KUKA KRL program: EPS_2_25694_WD06A_A_20260120031700.src

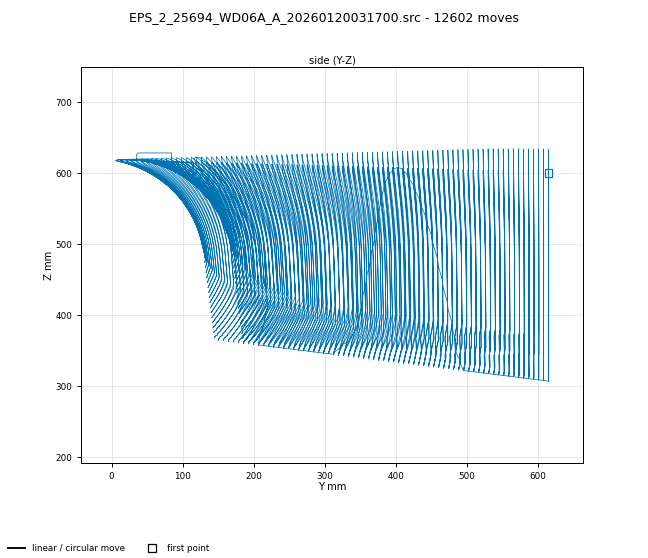
[picture p0: tool path of EPS_2_25694_WD06A_A_20260120031700.src, 12602 of 12604 moves have a stored position in this frame; points joined in program order, loops and branches not executed]
&ACCESS RVP
&REL 4
&COMMENT QRS 19112012
&PARAM EDITMASK = *
DEF PART()
EXT BAS (BAS_COMMAND :IN,REAL :IN )
INT I
BAS (#INITMOV,0 )

;KUKA QRS Post kuka4.cps  Date:22-06-2017 !

File_ID=2995

QRS_PRE_INIT()

;Init var - Until changes are made in qrs_pre_init
Outlet_Square_prg=0
Inlet_1_Square_prg=0
Inlet_2_Square_prg=0
Inlet_3_Square_prg=0
Inlet_4_Square_prg=0
Inlet_5_Square_prg=0

Outlet_1={X 0.000, Y 527.380, Z 509.000, B 0.000, E1 0.000 }
Inlet_1={X 0.000, Y 529.540, Z 479.000, B 0.000, E1 174.000 }
Outlet_1_type=251
Inlet_1_type=251
;QRS#1=Sidecore dimensions
;QRS#2=250-10" PVC SDR 35
;QRS#3=250-10" PVC SDR 35
;QRS#4=
;QRS#5=
;QRS#6=
;QRS#7=
;QRS#8=
;QRS#9=14M PSX
;QRS#10=14M PSX
;QRS#11=
;QRS#12=
;QRS#13=
;QRS#14=
;QRS#15=
;QRS#16=1220x127x914 3'
;QRS#17=EPS Height
;QRS#18=634,5
;QRS#19=*
;QRS#20= UPDATED VERSION 22-06-2017
;QRS#21=*
Outlet_Square=0100
Inlet_1_Square=0100
Inlet_2_Square=0
Inlet_3_Square=0
Inlet_4_Square=0
Inlet_5_Square=0
Mill_Square=1
Outlet_Square_Prg=205
Inlet_1_Square_prg=205

QRS_INIT()

$ADVANCE=5

; T1
PTP {E1 173.639,E2 173.639}
PTP {X 0,Y 615.429,A -85,B 0,C 180,E1 173.639,E2 173.639,E3 0,E4 0,E5 0,E6 0}
QRS_SPEED_INIT()
LIN {X 0,Y 615.429,Z 600,A -85,B 0,C 180,E1 173.639,E2 173.639,E3 0,E4 0,E5 0,E6 0} C_VEL
LIN {X 0,Y 615.429,Z 317.5,A -85,B 0,C 180,E1 173.639,E2 173.639} C_VEL
LIN {X 0,Y 615.429,Z 309.322,A -85,B 0,C 180,E1 173.639,E2 173.639} C_VEL
LIN {X 0,Y 615.432,Z 307.322,A -85,B 0,C 180,E1 173.453,E2 173.453} C_VEL
LIN {X 0,Y 615.494,Z 307.326,A -85,B 0,C 180,E1 170.801,E2 170.801} C_VEL
LIN {X 0,Y 615.451,Z 307.317,A -85,B 0,C 180,E1 168.138,E2 168.138} C_VEL
LIN {X 0,Y 615.446,Z 307.318,A -85,B 0,C 180,E1 166.077,E2 166.077} C_VEL
LIN {X 0,Y 615.443,Z 307.321,A -85,B 0,C 180,E1 163.578,E2 163.578} C_VEL
LIN {X 0,Y 615.461,Z 307.322,A -85,B 0,C 180,E1 161.353,E2 161.353} C_VEL
LIN {X 0,Y 615.492,Z 307.312,A -85,B 0,C 180,E1 158.568,E2 158.568} C_VEL
LIN {X 0,Y 615.449,Z 307.317,A -85,B 0,C 180,E1 155.996,E2 155.996} C_VEL
LIN {X 0,Y 615.462,Z 307.321,A -85,B 0,C 180,E1 153.554,E2 153.554} C_VEL
LIN {X 0,Y 615.485,Z 307.311,A -85,B 0,C 180,E1 150.593,E2 150.593} C_VEL
LIN {X 0,Y 615.466,Z 307.313,A -85,B 0,C 180,E1 148.313,E2 148.313} C_VEL
LIN {X 0,Y 615.458,Z 307.317,A -85,B 0,C 180,E1 145.976,E2 145.976} C_VEL
LIN {X 0,Y 615.49,Z 307.317,A -85,B 0,C 180,E1 143.061,E2 143.061} C_VEL
LIN {X 0,Y 615.465,Z 307.313,A -85,B 0,C 180,E1 140.248,E2 140.248} C_VEL
LIN {X 0,Y 615.481,Z 307.324,A -85,B 0,C 180,E1 137.646,E2 137.646} C_VEL
LIN {X 0,Y 615.484,Z 307.311,A -85,B 0,C 180,E1 134.93,E2 134.93} C_VEL
LIN {X 0,Y 615.469,Z 307.318,A -85,B 0,C 180,E1 132.078,E2 132.078} C_VEL
LIN {X 0,Y 615.491,Z 307.323,A -85,B 0,C 180,E1 129.748,E2 129.748} C_VEL
LIN {X 0,Y 615.484,Z 307.31,A -85,B 0,C 180,E1 126.935,E2 126.935} C_VEL
LIN {X 0,Y 615.491,Z 307.307,A -85,B 0,C 180,E1 124.7,E2 124.7} C_VEL
LIN {X 0,Y 615.477,Z 307.315,A -85,B 0,C 180,E1 122.328,E2 122.328} C_VEL
LIN {X 0,Y 615.495,Z 307.324,A -85,B 0,C 180,E1 119.795,E2 119.795} C_VEL
LIN {X 0,Y 615.485,Z 307.309,A -85,B 0,C 180,E1 117.043,E2 117.043} C_VEL
LIN {X 0,Y 615.484,Z 307.403,A -85,B 0,C 180,E1 116.593,E2 116.593} C_VEL
LIN {X 0,Y 615.488,Z 326.881,A -85,B 0,C 180,E1 113.782,E2 113.782} C_VEL
LIN {X 0,Y 615.482,Z 342.607,A -85,B 0,C 180,E1 111.541,E2 111.541} C_VEL
LIN {X 0,Y 615.492,Z 479.376,A -85,B 0,C 180,E1 109.902,E2 109.902} C_VEL
LIN {X 0,Y 615.495,Z 493.622,A -85,B 0,C 180,E1 109.597,E2 109.597} C_VEL
LIN {X 0,Y 615.494,Z 507.479,A -85,B 0,C 180,E1 109.164,E2 109.164} C_VEL
LIN {X 0,Y 615.498,Z 520.807,A -85,B 0,C 180,E1 108.606,E2 108.606} C_VEL
LIN {X 0,Y 615.497,Z 533.048,A -85,B 0,C 180,E1 107.956,E2 107.956} C_VEL
LIN {X 0,Y 615.497,Z 544.838,A -85,B 0,C 180,E1 107.184,E2 107.184} C_VEL
LIN {X 0,Y 615.497,Z 555.926,A -85,B 0,C 180,E1 106.3,E2 106.3} C_VEL
LIN {X 0,Y 615.497,Z 565.352,A -85,B 0,C 180,E1 105.395,E2 105.395} C_VEL
LIN {X 0,Y 615.497,Z 574.045,A -85,B 0,C 180,E1 104.395,E2 104.395} C_VEL
LIN {X 0,Y 615.496,Z 582.543,A -85,B 0,C 180,E1 103.201,E2 103.201} C_VEL
LIN {X 0,Y 615.495,Z 588.363,A -85,B 0,C 180,E1 102.195,E2 102.195} C_VEL
LIN {X 0,Y 615.497,Z 593.095,A -85,B 0,C 180,E1 101.193,E2 101.193} C_VEL
LIN {X 0,Y 615.497,Z 597.97,A -85,B 0,C 180,E1 99.862,E2 99.862} C_VEL
LIN {X 0,Y 615.494,Z 601.332,A -85,B 0,C 180,E1 98.536,E2 98.536} C_VEL
LIN {X 0,Y 615.493,Z 603.283,A -85,B 0,C 180,E1 97.215,E2 97.215} C_VEL
LIN {X 0,Y 615.497,Z 603.881,A -85,B 0,C 180,E1 95.898,E2 95.898} C_VEL
LIN {X 0,Y 615.491,Z 603.154,A -85,B 0,C 180,E1 94.584,E2 94.584} C_VEL
LIN {X 0,Y 615.492,Z 601.113,A -85,B 0,C 180,E1 93.273,E2 93.273} C_VEL
LIN {X 0,Y 615.499,Z 597.697,A -85,B 0,C 180,E1 91.963,E2 91.963} C_VEL
LIN {X 0,Y 615.495,Z 592.824,A -85,B 0,C 180,E1 90.654,E2 90.654} C_VEL
LIN {X 0,Y 615.494,Z 586.341,A -85,B 0,C 180,E1 89.346,E2 89.346} C_VEL
LIN {X 0,Y 615.496,Z 579.144,A -85,B 0,C 180,E1 88.201,E2 88.201} C_VEL
LIN {X 0,Y 615.495,Z 570.256,A -85,B 0,C 180,E1 87.055,E2 87.055} C_VEL
LIN {X 0,Y 615.496,Z 560.951,A -85,B 0,C 180,E1 86.072,E2 86.072} C_VEL
LIN {X 0,Y 615.498,Z 549.629,A -85,B 0,C 180,E1 85.087,E2 85.087} C_VEL
LIN {X 0,Y 615.497,Z 538.117,A -85,B 0,C 180,E1 84.266,E2 84.266} C_VEL
LIN {X 0,Y 615.491,Z 525.336,A -85,B 0,C 180,E1 83.526,E2 83.526} C_VEL
LIN {X 0,Y 615.493,Z 512.692,A -85,B 0,C 180,E1 82.945,E2 82.945} C_VEL
LIN {X 0,Y 615.494,Z 498.749,A -85,B 0,C 180,E1 82.455,E2 82.455} C_VEL
LIN {X 0,Y 615.493,Z 484.56,A -85,B 0,C 180,E1 82.104,E2 82.104} C_VEL
LIN {X 0,Y 615.487,Z 469.606,A -85,B 0,C 180,E1 81.877,E2 81.877} C_VEL
LIN {X 0,Y 615.485,Z 342.589,A -85,B 0,C 180,E1 80.366,E2 80.366} C_VEL
LIN {X 0,Y 615.494,Z 323.457,A -85,B 0,C 180,E1 77.638,E2 77.638} C_VEL
LIN {X 0,Y 615.487,Z 307.309,A -85,B 0,C 180,E1 75.282,E2 75.282} C_VEL
LIN {X 0,Y 615.477,Z 307.312,A -85,B 0,C 180,E1 72.73,E2 72.73} C_VEL
LIN {X 0,Y 615.486,Z 307.324,A -85,B 0,C 180,E1 69.968,E2 69.968} C_VEL
LIN {X 0,Y 615.486,Z 307.308,A -85,B 0,C 180,E1 67.156,E2 67.156} C_VEL
LIN {X 0,Y 615.494,Z 307.323,A -85,B 0,C 180,E1 64.285,E2 64.285} C_VEL
LIN {X 0,Y 615.472,Z 307.313,A -85,B 0,C 180,E1 61.553,E2 61.553} C_VEL
LIN {X 0,Y 615.486,Z 307.311,A -85,B 0,C 180,E1 58.915,E2 58.915} C_VEL
LIN {X 0,Y 615.473,Z 307.319,A -85,B 0,C 180,E1 55.978,E2 55.978} C_VEL
LIN {X 0,Y 615.472,Z 307.312,A -85,B 0,C 180,E1 53.575,E2 53.575} C_VEL
LIN {X 0,Y 615.488,Z 307.313,A -85,B 0,C 180,E1 50.939,E2 50.939} C_VEL
LIN {X 0,Y 615.494,Z 307.325,A -85,B 0,C 180,E1 48.528,E2 48.528} C_VEL
LIN {X 0,Y 615.461,Z 307.315,A -85,B 0,C 180,E1 45.85,E2 45.85} C_VEL
LIN {X 0,Y 615.492,Z 307.313,A -85,B 0,C 180,E1 43.05,E2 43.05} C_VEL
LIN {X 0,Y 615.483,Z 307.327,A -85,B 0,C 180,E1 40.607,E2 40.607} C_VEL
LIN {X 0,Y 615.454,Z 307.317,A -85,B 0,C 180,E1 38.01,E2 38.01} C_VEL
LIN {X 0,Y 615.468,Z 307.312,A -85,B 0,C 180,E1 35.618,E2 35.618} C_VEL
LIN {X 0,Y 615.493,Z 307.313,A -85,B 0,C 180,E1 33.236,E2 33.236} C_VEL
LIN {X 0,Y 615.497,Z 307.323,A -85,B 0,C 180,E1 30.92,E2 30.92} C_VEL
LIN {X 0,Y 615.456,Z 307.321,A -85,B 0,C 180,E1 28.448,E2 28.448} C_VEL
LIN {X 0,Y 615.451,Z 307.321,A -85,B 0,C 180,E1 26.446,E2 26.446} C_VEL
LIN {X 0,Y 615.444,Z 307.318,A -85,B 0,C 180,E1 24.003,E2 24.003} C_VEL
LIN {X 0,Y 615.491,Z 307.314,A -85,B 0,C 180,E1 21.432,E2 21.432} C_VEL
LIN {X 0,Y 615.447,Z 307.322,A -85,B 0,C 180,E1 18.598,E2 18.598} C_VEL
LIN {X 0,Y 615.435,Z 307.321,A -85,B 0,C 180,E1 16.42,E2 16.42} C_VEL
LIN {X 0,Y 615.437,Z 307.322,A -85,B 0,C 180,E1 14.551,E2 14.551} C_VEL
LIN {X 0,Y 615.433,Z 307.322,A -85,B 0,C 180,E1 12.532,E2 12.532} C_VEL
LIN {X 0,Y 615.43,Z 307.322,A -85,B 0,C 180,E1 10.528,E2 10.528} C_VEL
LIN {X 0,Y 615.427,Z 307.323,A -85,B 0,C 180,E1 8.538,E2 8.538} C_VEL
LIN {X 0,Y 615.424,Z 307.323,A -85,B 0,C 180,E1 6.541,E2 6.541} C_VEL
LIN {X 0,Y 615.422,Z 307.324,A -85,B 0,C 180,E1 4.585,E2 4.585} C_VEL
LIN {X 0,Y 615.421,Z 307.324,A -85,B 0,C 180,E1 2.618,E2 2.618} C_VEL
LIN {X 0,Y 615.419,Z 307.324,A -85,B 0,C 180,E1 0.655,E2 0.655} C_VEL
LIN {X 0,Y 615.417,Z 307.325,A -85,B 0,C 180,E1 -1.309,E2 -1.309} C_VEL
LIN {X 0,Y 615.415,Z 307.325,A -85,B 0,C 180,E1 -3.273,E2 -3.273} C_VEL
LIN {X 0,Y 615.415,Z 307.325,A -85,B 0,C 180,E1 -5.242,E2 -5.242} C_VEL
LIN {X 0,Y 615.418,Z 307.324,A -85,B 0,C 180,E1 -7.216,E2 -7.216} C_VEL
LIN {X 0,Y 615.42,Z 307.324,A -85,B 0,C 180,E1 -9.2,E2 -9.2} C_VEL
LIN {X 0,Y 615.421,Z 307.323,A -85,B 0,C 180,E1 -11.194,E2 -11.194} C_VEL
LIN {X 0,Y 615.423,Z 307.322,A -85,B 0,C 180,E1 -13.202,E2 -13.202} C_VEL
LIN {X 0,Y 615.422,Z 307.322,A -85,B 0,C 180,E1 -15.228,E2 -15.228} C_VEL
LIN {X 0,Y 615.425,Z 307.322,A -85,B 0,C 180,E1 -17.272,E2 -17.272} C_VEL
LIN {X 0,Y 615.48,Z 307.324,A -85,B 0,C 180,E1 -20.033,E2 -20.033} C_VEL
LIN {X 0,Y 615.446,Z 307.319,A -85,B 0,C 180,E1 -22.846,E2 -22.846} C_VEL
LIN {X 0,Y 615.438,Z 307.319,A -85,B 0,C 180,E1 -24.994,E2 -24.994} C_VEL
LIN {X 0,Y 615.436,Z 307.32,A -85,B 0,C 180,E1 -27.18,E2 -27.18} C_VEL
LIN {X 0,Y 615.476,Z 307.324,A -85,B 0,C 180,E1 -29.796,E2 -29.796} C_VEL
LIN {X 0,Y 615.482,Z 307.313,A -85,B 0,C 180,E1 -32.458,E2 -32.458} C_VEL
LIN {X 0,Y 615.451,Z 307.316,A -85,B 0,C 180,E1 -34.817,E2 -34.817} C_VEL
LIN {X 0,Y 615.448,Z 307.32,A -85,B 0,C 180,E1 -37.245,E2 -37.245} C_VEL
LIN {X 0,Y 615.494,Z 307.316,A -85,B 0,C 180,E1 -40.092,E2 -40.092} C_VEL
LIN {X 0,Y 615.489,Z 307.31,A -85,B 0,C 180,E1 -42.353,E2 -42.353} C_VEL
LIN {X 0,Y 615.454,Z 307.318,A -85,B 0,C 180,E1 -45.072,E2 -45.072} C_VEL
LIN {X 0,Y 615.492,Z 307.317,A -85,B 0,C 180,E1 -47.919,E2 -47.919} C_VEL
LIN {X 0,Y 615.493,Z 307.309,A -85,B 0,C 180,E1 -50.252,E2 -50.252} C_VEL
LIN {X 0,Y 615.463,Z 307.319,A -85,B 0,C 180,E1 -53.066,E2 -53.066} C_VEL
LIN {X 0,Y 615.481,Z 307.322,A -85,B 0,C 180,E1 -55.3,E2 -55.3} C_VEL
LIN {X 0,Y 615.484,Z 307.309,A -85,B 0,C 180,E1 -58.315,E2 -58.315} C_VEL
LIN {X 0,Y 615.469,Z 307.313,A -85,B 0,C 180,E1 -60.594,E2 -60.594} C_VEL
LIN {X 0,Y 615.472,Z 307.319,A -85,B 0,C 180,E1 -62.958,E2 -62.958} C_VEL
LIN {X 0,Y 615.483,Z 307.315,A -85,B 0,C 180,E1 -65.729,E2 -65.729} C_VEL
LIN {X 0,Y 615.474,Z 307.373,A -85,B 0,C 180,E1 -66.511,E2 -66.511} C_VEL
LIN {X 0,Y 615.496,Z 329.451,A -85,B 0,C 180,E1 -69.27,E2 -69.27} C_VEL
LIN {X 0,Y 615.498,Z 352.039,A -85,B 0,C 180,E1 -72.044,E2 -72.044} C_VEL
LIN {X 0,Y 615.49,Z 371.43,A -85,B 0,C 180,E1 -74.393,E2 -74.393} C_VEL
LIN {X 0,Y 615.498,Z 509.932,A -85,B 0,C 180,E1 -76.064,E2 -76.064} C_VEL
LIN {X 0,Y 615.495,Z 524.391,A -85,B 0,C 180,E1 -76.379,E2 -76.379} C_VEL
LIN {X 0,Y 615.489,Z 537.698,A -85,B 0,C 180,E1 -76.799,E2 -76.799} C_VEL
LIN {X 0,Y 615.498,Z 551.59,A -85,B 0,C 180,E1 -77.387,E2 -77.387} C_VEL
LIN {X 0,Y 615.495,Z 564.013,A -85,B 0,C 180,E1 -78.056,E2 -78.056} C_VEL
LIN {X 0,Y 615.499,Z 575.344,A -85,B 0,C 180,E1 -78.807,E2 -78.807} C_VEL
LIN {X 0,Y 615.498,Z 585.752,A -85,B 0,C 180,E1 -79.64,E2 -79.64} C_VEL
LIN {X 0,Y 615.496,Z 596.091,A -85,B 0,C 180,E1 -80.636,E2 -80.636} C_VEL
LIN {X 0,Y 615.497,Z 604.605,A -85,B 0,C 180,E1 -81.629,E2 -81.629} C_VEL
LIN {X 0,Y 615.496,Z 612.728,A -85,B 0,C 180,E1 -82.785,E2 -82.785} C_VEL
LIN {X 0,Y 615.496,Z 618.431,A -85,B 0,C 180,E1 -83.773,E2 -83.773} C_VEL
LIN {X 0,Y 615.495,Z 623.081,A -85,B 0,C 180,E1 -84.759,E2 -84.759} C_VEL
LIN {X 0,Y 615.494,Z 627.902,A -85,B 0,C 180,E1 -86.072,E2 -86.072} C_VEL
LIN {X 0,Y 615.496,Z 631.252,A -85,B 0,C 180,E1 -87.382,E2 -87.382} C_VEL
LIN {X 0,Y 615.489,Z 633.229,A -85,B 0,C 180,E1 -88.691,E2 -88.691} C_VEL
LIN {X 0,Y 615.493,Z 633.889,A -85,B 0,C 180,E1 -90,E2 -90} C_VEL
LIN {X 0,Y 615.489,Z 633.229,A -85,B 0,C 180,E1 -91.309,E2 -91.309} C_VEL
LIN {X 0,Y 615.496,Z 631.252,A -85,B 0,C 180,E1 -92.618,E2 -92.618} C_VEL
LIN {X 0,Y 615.494,Z 627.902,A -85,B 0,C 180,E1 -93.928,E2 -93.928} C_VEL
LIN {X 0,Y 615.495,Z 623.081,A -85,B 0,C 180,E1 -95.241,E2 -95.241} C_VEL
LIN {X 0,Y 615.496,Z 616.629,A -85,B 0,C 180,E1 -96.556,E2 -96.556} C_VEL
LIN {X 0,Y 615.497,Z 609.442,A -85,B 0,C 180,E1 -97.71,E2 -97.71} C_VEL
LIN {X 0,Y 615.497,Z 601.905,A -85,B 0,C 180,E1 -98.702,E2 -98.702} C_VEL
LIN {X 0,Y 615.495,Z 592.855,A -85,B 0,C 180,E1 -99.696,E2 -99.696} C_VEL
LIN {X 0,Y 615.497,Z 582.76,A -85,B 0,C 180,E1 -100.618,E2 -100.618} C_VEL
LIN {X 0,Y 615.498,Z 571.861,A -85,B 0,C 180,E1 -101.443,E2 -101.443} C_VEL
LIN {X 0,Y 615.489,Z 559.711,A -85,B 0,C 180,E1 -102.195,E2 -102.195} C_VEL
LIN {X 0,Y 615.498,Z 546.097,A -85,B 0,C 180,E1 -102.865,E2 -102.865} C_VEL
LIN {X 0,Y 615.49,Z 532.845,A -85,B 0,C 180,E1 -103.369,E2 -103.369} C_VEL
LIN {X 0,Y 615.494,Z 519.301,A -85,B 0,C 180,E1 -103.747,E2 -103.747} C_VEL
LIN {X 0,Y 615.494,Z 504.744,A -85,B 0,C 180,E1 -104.013,E2 -104.013} C_VEL
LIN {X 0,Y 615.49,Z 371.43,A -85,B 0,C 180,E1 -105.607,E2 -105.607} C_VEL
LIN {X 0,Y 615.485,Z 348.061,A -85,B 0,C 180,E1 -108.442,E2 -108.442} C_VEL
LIN {X 0,Y 615.489,Z 325.212,A -85,B 0,C 180,E1 -111.256,E2 -111.256} C_VEL
LIN {X 0,Y 615.475,Z 307.311,A -85,B 0,C 180,E1 -113.512,E2 -113.512} C_VEL
LIN {X 0,Y 615.483,Z 307.321,A -85,B 0,C 180,E1 -116.444,E2 -116.444} C_VEL
LIN {X 0,Y 615.484,Z 307.327,A -85,B 0,C 180,E1 -118.657,E2 -118.657} C_VEL
LIN {X 0,Y 615.464,Z 307.318,A -85,B 0,C 180,E1 -121.082,E2 -121.082} C_VEL
LIN {X 0,Y 615.474,Z 307.311,A -85,B 0,C 180,E1 -123.532,E2 -123.532} C_VEL
LIN {X 0,Y 615.484,Z 307.327,A -85,B 0,C 180,E1 -126.424,E2 -126.424} C_VEL
LIN {X 0,Y 615.457,Z 307.317,A -85,B 0,C 180,E1 -129.059,E2 -129.059} C_VEL
LIN {X 0,Y 615.47,Z 307.312,A -85,B 0,C 180,E1 -131.474,E2 -131.474} C_VEL
LIN {X 0,Y 615.494,Z 307.321,A -85,B 0,C 180,E1 -134.147,E2 -134.147} C_VEL
LIN {X 0,Y 615.455,Z 307.32,A -85,B 0,C 180,E1 -136.753,E2 -136.753} C_VEL
LIN {X 0,Y 615.464,Z 307.314,A -85,B 0,C 180,E1 -139.392,E2 -139.392} C_VEL
LIN {X 0,Y 615.491,Z 307.321,A -85,B 0,C 180,E1 -141.986,E2 -141.986} C_VEL
LIN {X 0,Y 615.464,Z 307.323,A -85,B 0,C 180,E1 -144.383,E2 -144.383} C_VEL
LIN {X 0,Y 615.44,Z 307.32,A -85,B 0,C 180,E1 -146.761,E2 -146.761} C_VEL
LIN {X 0,Y 615.442,Z 307.318,A -85,B 0,C 180,E1 -149.078,E2 -149.078} C_VEL
LIN {X 0,Y 615.484,Z 307.316,A -85,B 0,C 180,E1 -151.547,E2 -151.547} C_VEL
LIN {X 0,Y 615.441,Z 307.322,A -85,B 0,C 180,E1 -154.437,E2 -154.437} C_VEL
LIN {X 0,Y 615.436,Z 307.323,A -85,B 0,C 180,E1 -156.442,E2 -156.442} C_VEL
LIN {X 0,Y 615.428,Z 307.322,A -85,B 0,C 180,E1 -158.566,E2 -158.566} C_VEL
LIN {X 0,Y 615.423,Z 307.322,A -85,B 0,C 180,E1 -160.66,E2 -160.66} C_VEL
LIN {X 0,Y 615.47,Z 307.322,A -85,B 0,C 180,E1 -163.413,E2 -163.413} C_VEL
LIN {X 0,Y 615.438,Z 307.324,A -85,B 0,C 180,E1 -166.125,E2 -166.125} C_VEL
LIN {X 0,Y 615.432,Z 307.325,A -85,B 0,C 180,E1 -168.138,E2 -168.138} C_VEL
LIN {X 0,Y 615.428,Z 307.325,A -85,B 0,C 180,E1 -170.137,E2 -170.137} C_VEL
LIN {X 0,Y 615.426,Z 307.325,A -85,B 0,C 180,E1 -172.124,E2 -172.124} C_VEL
LIN {X 0,Y 615.429,Z 307.324,A -85,B 0,C 180,E1 -174.101,E2 -174.101} C_VEL
LIN {X 0,Y 615.431,Z 307.323,A -85,B 0,C 180,E1 -176.071,E2 -176.071} C_VEL
LIN {X 0,Y 615.435,Z 307.322,A -85,B 0,C 180,E1 -178.037,E2 -178.037} C_VEL
LIN {X 0,Y 615.437,Z 307.322,A -85,B 0,C 180,E1 -180,E2 -180} C_VEL
LIN {X 0,Y 615.441,Z 307.321,A -85,B 0,C 180,E1 -181.963,E2 -181.963} C_VEL
LIN {X 0,Y 615.443,Z 307.32,A -85,B 0,C 180,E1 -183.929,E2 -183.929} C_VEL
LIN {X 0,Y 615.447,Z 307.319,A -85,B 0,C 180,E1 -185.899,E2 -185.899} C_VEL
LIN {X 0,Y 615.432,Z 307.322,A -85,B 0,C 180,E1 -186.547,E2 -186.547} C_VEL
LIN {X 0,Y 614.801,Z 307.472,A -85,B 0,C 180,E1 -187.093,E2 -187.093} C_VEL
LIN {X 0,Y 612.004,Z 307.871,A -85,B 0,C 180,E1 -187.98,E2 -187.98} C_VEL
LIN {X 0,Y 609.609,Z 308.187,A -85,B 0,C 180,E1 -188.692,E2 -188.692} C_VEL
LIN {X 0,Y 608.553,Z 308.31,A -85,B 0,C 180,E1 -189.242,E2 -189.242} C_VEL
LIN {X 0,Y 608.454,Z 308.318,A -85,B 0,C 180,E1 -189.428,E2 -189.428} C_VEL
LIN {X 0,Y 608.428,Z 308.316,A -85,B 0,C 180,E1 -192.001,E2 -192.001} C_VEL
LIN {X 0,Y 608.43,Z 308.315,A -85,B 0,C 180,E1 -194.039,E2 -194.039} C_VEL
LIN {X 0,Y 608.439,Z 308.317,A -85,B 0,C 180,E1 -196.525,E2 -196.525} C_VEL
LIN {X 0,Y 608.439,Z 308.316,A -85,B 0,C 180,E1 -199.571,E2 -199.571} C_VEL
LIN {X 0,Y 608.456,Z 308.313,A -85,B 0,C 180,E1 -201.692,E2 -201.692} C_VEL
LIN {X 0,Y 608.437,Z 308.32,A -85,B 0,C 180,E1 -204.572,E2 -204.572} C_VEL
LIN {X 0,Y 608.48,Z 308.313,A -85,B 0,C 180,E1 -207.211,E2 -207.211} C_VEL
LIN {X 0,Y 608.441,Z 308.314,A -85,B 0,C 180,E1 -209.97,E2 -209.97} C_VEL
LIN {X 0,Y 608.45,Z 308.32,A -85,B 0,C 180,E1 -212.523,E2 -212.523} C_VEL
LIN {X 0,Y 608.437,Z 308.316,A -85,B 0,C 180,E1 -215.279,E2 -215.279} C_VEL
LIN {X 0,Y 608.455,Z 308.312,A -85,B 0,C 180,E1 -217.748,E2 -217.748} C_VEL
LIN {X 0,Y 608.443,Z 308.32,A -85,B 0,C 180,E1 -220.33,E2 -220.33} C_VEL
LIN {X 0,Y 608.482,Z 308.309,A -85,B 0,C 180,E1 -223.312,E2 -223.312} C_VEL
LIN {X 0,Y 608.458,Z 308.317,A -85,B 0,C 180,E1 -226.131,E2 -226.131} C_VEL
LIN {X 0,Y 608.455,Z 308.316,A -85,B 0,C 180,E1 -228.825,E2 -228.825} C_VEL
LIN {X 0,Y 608.467,Z 308.311,A -85,B 0,C 180,E1 -231.413,E2 -231.413} C_VEL
LIN {X 0,Y 608.446,Z 308.318,A -85,B 0,C 180,E1 -233.955,E2 -233.955} C_VEL
LIN {X 0,Y 608.466,Z 308.32,A -85,B 0,C 180,E1 -236.33,E2 -236.33} C_VEL
LIN {X 0,Y 608.447,Z 308.315,A -85,B 0,C 180,E1 -238.733,E2 -238.733} C_VEL
LIN {X 0,Y 608.47,Z 308.311,A -85,B 0,C 180,E1 -241.382,E2 -241.382} C_VEL
LIN {X 0,Y 608.492,Z 308.363,A -85,B 0,C 180,E1 -243.298,E2 -243.298} C_VEL
LIN {X 0,Y 608.515,Z 326.387,A -85,B 0,C 180,E1 -245.929,E2 -245.929} C_VEL
LIN {X 0,Y 608.501,Z 342.709,A -85,B 0,C 180,E1 -248.277,E2 -248.277} C_VEL
LIN {X 0,Y 608.628,Z 478.925,A -85,B 0,C 180,E1 -249.93,E2 -249.93} C_VEL
LIN {X 0,Y 608.606,Z 493.353,A -85,B 0,C 180,E1 -250.238,E2 -250.238} C_VEL
LIN {X 0,Y 608.58,Z 506.716,A -85,B 0,C 180,E1 -250.654,E2 -250.654} C_VEL
LIN {X 0,Y 608.556,Z 519.861,A -85,B 0,C 180,E1 -251.199,E2 -251.199} C_VEL
LIN {X 0,Y 608.516,Z 531.906,A -85,B 0,C 180,E1 -251.831,E2 -251.831} C_VEL
LIN {X 0,Y 608.527,Z 543.965,A -85,B 0,C 180,E1 -252.613,E2 -252.613} C_VEL
LIN {X 0,Y 608.482,Z 554.83,A -85,B 0,C 180,E1 -253.468,E2 -253.468} C_VEL
LIN {X 0,Y 608.471,Z 564.893,A -85,B 0,C 180,E1 -254.423,E2 -254.423} C_VEL
LIN {X 0,Y 608.457,Z 573.894,A -85,B 0,C 180,E1 -255.45,E2 -255.45} C_VEL
LIN {X 0,Y 608.457,Z 581.334,A -85,B 0,C 180,E1 -256.474,E2 -256.474} C_VEL
LIN {X 0,Y 608.456,Z 588.411,A -85,B 0,C 180,E1 -257.662,E2 -257.662} C_VEL
LIN {X 0,Y 608.429,Z 593.28,A -85,B 0,C 180,E1 -258.676,E2 -258.676} C_VEL
LIN {X 0,Y 608.437,Z 598.287,A -85,B 0,C 180,E1 -260.023,E2 -260.023} C_VEL
LIN {X 0,Y 608.419,Z 601.76,A -85,B 0,C 180,E1 -261.364,E2 -261.364} C_VEL
LIN {X 0,Y 608.42,Z 603.806,A -85,B 0,C 180,E1 -262.7,E2 -262.7} C_VEL
LIN {X 0,Y 608.433,Z 604.5,A -85,B 0,C 180,E1 -264.033,E2 -264.033} C_VEL
LIN {X 0,Y 608.425,Z 603.838,A -85,B 0,C 180,E1 -265.362,E2 -265.362} C_VEL
LIN {X 0,Y 608.42,Z 601.84,A -85,B 0,C 180,E1 -266.689,E2 -266.689} C_VEL
LIN {X 0,Y 608.444,Z 598.457,A -85,B 0,C 180,E1 -268.014,E2 -268.014} C_VEL
LIN {X 0,Y 608.439,Z 593.606,A -85,B 0,C 180,E1 -269.338,E2 -269.338} C_VEL
LIN {X 0,Y 608.438,Z 587.139,A -85,B 0,C 180,E1 -270.662,E2 -270.662} C_VEL
LIN {X 0,Y 608.444,Z 579.966,A -85,B 0,C 180,E1 -271.82,E2 -271.82} C_VEL
LIN {X 0,Y 608.482,Z 571.13,A -85,B 0,C 180,E1 -272.979,E2 -272.979} C_VEL
LIN {X 0,Y 608.471,Z 561.9,A -85,B 0,C 180,E1 -273.974,E2 -273.974} C_VEL
LIN {X 0,Y 608.501,Z 550.66,A -85,B 0,C 180,E1 -274.969,E2 -274.969} C_VEL
LIN {X 0,Y 608.519,Z 539.276,A -85,B 0,C 180,E1 -275.8,E2 -275.8} C_VEL
LIN {X 0,Y 608.526,Z 526.693,A -85,B 0,C 180,E1 -276.549,E2 -276.549} C_VEL
LIN {X 0,Y 608.551,Z 514.466,A -85,B 0,C 180,E1 -277.131,E2 -277.131} C_VEL
LIN {X 0,Y 608.574,Z 500.947,A -85,B 0,C 180,E1 -277.632,E2 -277.632} C_VEL
LIN {X 0,Y 608.604,Z 486.913,A -85,B 0,C 180,E1 -278.007,E2 -278.007} C_VEL
LIN {X 0,Y 608.626,Z 473.539,A -85,B 0,C 180,E1 -278.236,E2 -278.236} C_VEL
LIN {X 0,Y 608.498,Z 342.743,A -85,B 0,C 180,E1 -279.808,E2 -279.808} C_VEL
LIN {X 0,Y 608.533,Z 324.002,A -85,B 0,C 180,E1 -282.506,E2 -282.506} C_VEL
LIN {X 0,Y 608.481,Z 308.311,A -85,B 0,C 180,E1 -284.805,E2 -284.805} C_VEL
LIN {X 0,Y 608.45,Z 308.316,A -85,B 0,C 180,E1 -287.476,E2 -287.476} C_VEL
LIN {X 0,Y 608.46,Z 308.316,A -85,B 0,C 180,E1 -290.274,E2 -290.274} C_VEL
LIN {X 0,Y 608.45,Z 308.314,A -85,B 0,C 180,E1 -293.123,E2 -293.123} C_VEL
LIN {X 0,Y 608.475,Z 308.319,A -85,B 0,C 180,E1 -295.72,E2 -295.72} C_VEL
LIN {X 0,Y 608.442,Z 308.316,A -85,B 0,C 180,E1 -298.266,E2 -298.266} C_VEL
LIN {X 0,Y 608.468,Z 308.311,A -85,B 0,C 180,E1 -300.544,E2 -300.544} C_VEL
LIN {X 0,Y 608.453,Z 308.313,A -85,B 0,C 180,E1 -302.879,E2 -302.879} C_VEL
LIN {X 0,Y 608.454,Z 308.317,A -85,B 0,C 180,E1 -305.276,E2 -305.276} C_VEL
LIN {X 0,Y 608.459,Z 308.319,A -85,B 0,C 180,E1 -307.746,E2 -307.746} C_VEL
LIN {X 0,Y 608.436,Z 308.315,A -85,B 0,C 180,E1 -310.327,E2 -310.327} C_VEL
LIN {X 0,Y 608.453,Z 308.315,A -85,B 0,C 180,E1 -312.958,E2 -312.958} C_VEL
LIN {X 0,Y 608.437,Z 308.319,A -85,B 0,C 180,E1 -315.736,E2 -315.736} C_VEL
LIN {X 0,Y 608.441,Z 308.316,A -85,B 0,C 180,E1 -317.936,E2 -317.936} C_VEL
LIN {X 0,Y 608.443,Z 308.315,A -85,B 0,C 180,E1 -320.704,E2 -320.704} C_VEL
LIN {X 0,Y 608.457,Z 308.319,A -85,B 0,C 180,E1 -323.085,E2 -323.085} C_VEL
LIN {X 0,Y 608.46,Z 308.317,A -85,B 0,C 180,E1 -325.53,E2 -325.53} C_VEL
LIN {X 0,Y 608.44,Z 308.315,A -85,B 0,C 180,E1 -327.904,E2 -327.904} C_VEL
LIN {X 0,Y 608.44,Z 308.314,A -85,B 0,C 180,E1 -330.219,E2 -330.219} C_VEL
LIN {X 0,Y 608.482,Z 308.314,A -85,B 0,C 180,E1 -332.789,E2 -332.789} C_VEL
LIN {X 0,Y 608.433,Z 308.319,A -85,B 0,C 180,E1 -335.428,E2 -335.428} C_VEL
LIN {X 0,Y 608.454,Z 308.313,A -85,B 0,C 180,E1 -338.308,E2 -338.308} C_VEL
LIN {X 0,Y 608.443,Z 308.318,A -85,B 0,C 180,E1 -341.287,E2 -341.287} C_VEL
LIN {X 0,Y 608.417,Z 308.317,A -85,B 0,C 180,E1 -343.905,E2 -343.905} C_VEL
LIN {X 0,Y 608.46,Z 308.319,A -85,B 0,C 180,E1 -346.643,E2 -346.643} C_VEL
LIN {X 0,Y 608.419,Z 308.318,A -85,B 0,C 180,E1 -349.349,E2 -349.349} C_VEL
LIN {X 0,Y 608.411,Z 308.319,A -85,B 0,C 180,E1 -351.363,E2 -351.363} C_VEL
LIN {X 0,Y 608.421,Z 308.317,A -85,B 0,C 180,E1 -353.401,E2 -353.401} C_VEL
LIN {X 0,Y 608.396,Z 308.32,A -85,B 0,C 180,E1 -355.362,E2 -355.362} C_VEL
LIN {X 0,Y 608.418,Z 308.317,A -85,B 0,C 180,E1 -357.351,E2 -357.351} C_VEL
LIN {X 0,Y 608.397,Z 308.32,A -85,B 0,C 180,E1 -359.338,E2 -359.338} C_VEL
LIN {X 0,Y 608.406,Z 308.319,A -85,B 0,C 180,E1 -361.324,E2 -361.324} C_VEL
LIN {X 0,Y 608.385,Z 308.321,A -85,B 0,C 180,E1 -363.311,E2 -363.311} C_VEL
LIN {X 0,Y 608.399,Z 308.319,A -85,B 0,C 180,E1 -365.302,E2 -365.302} C_VEL
LIN {X 0,Y 608.395,Z 308.32,A -85,B 0,C 180,E1 -367.3,E2 -367.3} C_VEL
LIN {X 0,Y 608.416,Z 308.321,A -85,B 0,C 180,E1 -369.978,E2 -369.978} C_VEL
LIN {X 0,Y 608.454,Z 308.317,A -85,B 0,C 180,E1 -372.677,E2 -372.677} C_VEL
LIN {X 0,Y 608.418,Z 308.317,A -85,B 0,C 180,E1 -375.407,E2 -375.407} C_VEL
LIN {X 0,Y 608.406,Z 308.319,A -85,B 0,C 180,E1 -377.478,E2 -377.478} C_VEL
LIN {X 0,Y 608.414,Z 308.319,A -85,B 0,C 180,E1 -379.572,E2 -379.572} C_VEL
LIN {X 0,Y 608.463,Z 308.317,A -85,B 0,C 180,E1 -382.406,E2 -382.406} C_VEL
LIN {X 0,Y 608.438,Z 308.317,A -85,B 0,C 180,E1 -384.572,E2 -384.572} C_VEL
LIN {X 0,Y 608.415,Z 308.317,A -85,B 0,C 180,E1 -387.199,E2 -387.199} C_VEL
LIN {X 0,Y 608.463,Z 308.322,A -85,B 0,C 180,E1 -389.974,E2 -389.974} C_VEL
LIN {X 0,Y 608.434,Z 308.315,A -85,B 0,C 180,E1 -392.881,E2 -392.881} C_VEL
LIN {X 0,Y 608.42,Z 308.318,A -85,B 0,C 180,E1 -395.279,E2 -395.279} C_VEL
LIN {X 0,Y 608.466,Z 308.314,A -85,B 0,C 180,E1 -398.242,E2 -398.242} C_VEL
LIN {X 0,Y 608.438,Z 308.318,A -85,B 0,C 180,E1 -401.342,E2 -401.342} C_VEL
LIN {X 0,Y 608.459,Z 308.314,A -85,B 0,C 180,E1 -404.266,E2 -404.266} C_VEL
LIN {X 0,Y 608.425,Z 308.318,A -85,B 0,C 180,E1 -407.039,E2 -407.039} C_VEL
LIN {X 0,Y 608.451,Z 308.322,A -85,B 0,C 180,E1 -409.698,E2 -409.698} C_VEL
LIN {X 0,Y 608.465,Z 308.312,A -85,B 0,C 180,E1 -412.255,E2 -412.255} C_VEL
LIN {X 0,Y 608.435,Z 308.315,A -85,B 0,C 180,E1 -414.723,E2 -414.723} C_VEL
LIN {X 0,Y 608.464,Z 308.322,A -85,B 0,C 180,E1 -417.477,E2 -417.477} C_VEL
LIN {X 0,Y 608.48,Z 308.309,A -85,B 0,C 180,E1 -420.222,E2 -420.222} C_VEL
LIN {X 0,Y 608.465,Z 308.313,A -85,B 0,C 180,E1 -422.795,E2 -422.795} C_VEL
LIN {X 0,Y 608.448,Z 308.323,A -85,B 0,C 180,E1 -425.429,E2 -425.429} C_VEL
LIN {X 0,Y 608.48,Z 308.433,A -85,B 0,C 180,E1 -426.36,E2 -426.36} C_VEL
LIN {X 0,Y 608.595,Z 325.212,A -85,B 0,C 180,E1 -428.492,E2 -428.492} C_VEL
LIN {X 0,Y 608.535,Z 347.483,A -85,B 0,C 180,E1 -431.267,E2 -431.267} C_VEL
LIN {X 0,Y 608.516,Z 371.136,A -85,B 0,C 180,E1 -434.166,E2 -434.166} C_VEL
LIN {X 0,Y 608.571,Z 372.077,A -85,B 0,C 180,E1 -434.232,E2 -434.232} C_VEL
LIN {X 0,Y 608.615,Z 509.919,A -85,B 0,C 180,E1 -435.903,E2 -435.903} C_VEL
LIN {X 0,Y 608.598,Z 524.398,A -85,B 0,C 180,E1 -436.222,E2 -436.222} C_VEL
LIN {X 0,Y 608.579,Z 537.72,A -85,B 0,C 180,E1 -436.647,E2 -436.647} C_VEL
LIN {X 0,Y 608.565,Z 549.89,A -85,B 0,C 180,E1 -437.156,E2 -437.156} C_VEL
LIN {X 0,Y 608.516,Z 562.686,A -85,B 0,C 180,E1 -437.832,E2 -437.832} C_VEL
LIN {X 0,Y 608.499,Z 575.475,A -85,B 0,C 180,E1 -438.677,E2 -438.677} C_VEL
LIN {X 0,Y 608.496,Z 585.934,A -85,B 0,C 180,E1 -439.519,E2 -439.519} C_VEL
LIN {X 0,Y 608.479,Z 596.337,A -85,B 0,C 180,E1 -440.527,E2 -440.527} C_VEL
LIN {X 0,Y 608.464,Z 604.916,A -85,B 0,C 180,E1 -441.532,E2 -441.532} C_VEL
LIN {X 0,Y 608.461,Z 613.115,A -85,B 0,C 180,E1 -442.701,E2 -442.701} C_VEL
LIN {X 0,Y 608.443,Z 619.546,A -85,B 0,C 180,E1 -443.831,E2 -443.831} C_VEL
LIN {X 0,Y 608.438,Z 624.962,A -85,B 0,C 180,E1 -445.03,E2 -445.03} C_VEL
LIN {X 0,Y 608.431,Z 628.442,A -85,B 0,C 180,E1 -446.026,E2 -446.026} C_VEL
LIN {X 0,Y 608.424,Z 631.831,A -85,B 0,C 180,E1 -447.352,E2 -447.352} C_VEL
LIN {X 0,Y 608.442,Z 633.83,A -85,B 0,C 180,E1 -448.676,E2 -448.676} C_VEL
LIN {X 0,Y 608.433,Z 634.5,A -85,B 0,C 180,E1 -450,E2 -450} C_VEL
LIN {X 0,Y 608.442,Z 633.83,A -85,B 0,C 180,E1 -451.324,E2 -451.324} C_VEL
LIN {X 0,Y 608.424,Z 631.831,A -85,B 0,C 180,E1 -452.648,E2 -452.648} C_VEL
LIN {X 0,Y 608.431,Z 628.442,A -85,B 0,C 180,E1 -453.974,E2 -453.974} C_VEL
LIN {X 0,Y 608.44,Z 623.568,A -85,B 0,C 180,E1 -455.302,E2 -455.302} C_VEL
LIN {X 0,Y 608.445,Z 617.212,A -85,B 0,C 180,E1 -456.603,E2 -456.603} C_VEL
LIN {X 0,Y 608.453,Z 609.799,A -85,B 0,C 180,E1 -457.8,E2 -457.8} C_VEL
LIN {X 0,Y 608.473,Z 600.825,A -85,B 0,C 180,E1 -458.97,E2 -458.97} C_VEL
LIN {X 0,Y 608.472,Z 591.393,A -85,B 0,C 180,E1 -459.977,E2 -459.977} C_VEL
LIN {X 0,Y 608.505,Z 580.049,A -85,B 0,C 180,E1 -460.973,E2 -460.973} C_VEL
LIN {X 0,Y 608.533,Z 568.152,A -85,B 0,C 180,E1 -461.829,E2 -461.829} C_VEL
LIN {X 0,Y 608.531,Z 555.078,A -85,B 0,C 180,E1 -462.591,E2 -462.591} C_VEL
LIN {X 0,Y 608.556,Z 542.18,A -85,B 0,C 180,E1 -463.184,E2 -463.184} C_VEL
LIN {X 0,Y 608.593,Z 528.193,A -85,B 0,C 180,E1 -463.672,E2 -463.672} C_VEL
LIN {X 0,Y 608.621,Z 514.471,A -85,B 0,C 180,E1 -464.012,E2 -464.012} C_VEL
LIN {X 0,Y 608.621,Z 498.193,A -85,B 0,C 180,E1 -464.257,E2 -464.257} C_VEL
LIN {X 0,Y 608.53,Z 371.577,A -85,B 0,C 180,E1 -465.78,E2 -465.78} C_VEL
LIN {X 0,Y 608.567,Z 346.408,A -85,B 0,C 180,E1 -468.865,E2 -468.865} C_VEL
LIN {X 0,Y 608.596,Z 323.799,A -85,B 0,C 180,E1 -471.686,E2 -471.686} C_VEL
LIN {X 0,Y 608.473,Z 308.344,A -85,B 0,C 180,E1 -473.652,E2 -473.652} C_VEL
LIN {X 0,Y 608.445,Z 308.315,A -85,B 0,C 180,E1 -476.035,E2 -476.035} C_VEL
LIN {X 0,Y 608.473,Z 308.321,A -85,B 0,C 180,E1 -478.62,E2 -478.62} C_VEL
LIN {X 0,Y 608.439,Z 308.315,A -85,B 0,C 180,E1 -481.317,E2 -481.317} C_VEL
LIN {X 0,Y 608.468,Z 308.311,A -85,B 0,C 180,E1 -483.734,E2 -483.734} C_VEL
LIN {X 0,Y 608.475,Z 308.314,A -85,B 0,C 180,E1 -486.089,E2 -486.089} C_VEL
LIN {X 0,Y 608.456,Z 308.32,A -85,B 0,C 180,E1 -488.588,E2 -488.588} C_VEL
LIN {X 0,Y 608.441,Z 308.314,A -85,B 0,C 180,E1 -491.34,E2 -491.34} C_VEL
LIN {X 0,Y 608.472,Z 308.313,A -85,B 0,C 180,E1 -493.868,E2 -493.868} C_VEL
LIN {X 0,Y 608.447,Z 308.317,A -85,B 0,C 180,E1 -496.692,E2 -496.692} C_VEL
LIN {X 0,Y 608.421,Z 308.318,A -85,B 0,C 180,E1 -498.821,E2 -498.821} C_VEL
LIN {X 0,Y 608.465,Z 308.315,A -85,B 0,C 180,E1 -501.758,E2 -501.758} C_VEL
LIN {X 0,Y 608.471,Z 308.318,A -85,B 0,C 180,E1 -503.949,E2 -503.949} C_VEL
LIN {X 0,Y 608.432,Z 308.321,A -85,B 0,C 180,E1 -506.327,E2 -506.327} C_VEL
LIN {X 0,Y 608.423,Z 308.317,A -85,B 0,C 180,E1 -508.734,E2 -508.734} C_VEL
LIN {X 0,Y 608.458,Z 308.313,A -85,B 0,C 180,E1 -511.38,E2 -511.38} C_VEL
LIN {X 0,Y 608.438,Z 308.318,A -85,B 0,C 180,E1 -514.282,E2 -514.282} C_VEL
LIN {X 0,Y 608.447,Z 308.319,A -85,B 0,C 180,E1 -516.154,E2 -516.154} C_VEL
LIN {X 0,Y 608.435,Z 308.317,A -85,B 0,C 180,E1 -518.307,E2 -518.307} C_VEL
LIN {X 0,Y 608.409,Z 308.319,A -85,B 0,C 180,E1 -520.428,E2 -520.428} C_VEL
LIN {X 0,Y 608.419,Z 308.319,A -85,B 0,C 180,E1 -523.215,E2 -523.215} C_VEL
LIN {X 0,Y 608.416,Z 308.322,A -85,B 0,C 180,E1 -525.997,E2 -525.997} C_VEL
LIN {X 0,Y 608.42,Z 308.32,A -85,B 0,C 180,E1 -528,E2 -528} C_VEL
LIN {X 0,Y 608.41,Z 308.321,A -85,B 0,C 180,E1 -530.022,E2 -530.022} C_VEL
LIN {X 0,Y 608.394,Z 308.32,A -85,B 0,C 180,E1 -532.7,E2 -532.7} C_VEL
LIN {X 0,Y 608.454,Z 308.321,A -85,B 0,C 180,E1 -535.363,E2 -535.363} C_VEL
LIN {X 0,Y 608.408,Z 308.32,A -85,B 0,C 180,E1 -538.014,E2 -538.014} C_VEL
LIN {X 0,Y 608.431,Z 308.317,A -85,B 0,C 180,E1 -540,E2 -540} C_VEL
LIN {X 0,Y 608.412,Z 308.319,A -85,B 0,C 180,E1 -541.986,E2 -541.986} C_VEL
LIN {X 0,Y 608.411,Z 308.319,A -85,B 0,C 180,E1 -543.975,E2 -543.975} C_VEL
LIN {X 0,Y 608.421,Z 308.317,A -85,B 0,C 180,E1 -545.968,E2 -545.968} C_VEL
LIN {X 0,Y 608.414,Z 308.318,A -85,B 0,C 180,E1 -547.968,E2 -547.968} C_VEL
LIN {X 0,Y 608.454,Z 308.318,A -85,B 0,C 180,E1 -549.428,E2 -549.428} C_VEL
LIN {X 0,Y 607.751,Z 308.402,A -85,B 0,C 180,E1 -549.981,E2 -549.981} C_VEL
LIN {X 0,Y 604.885,Z 308.763,A -85,B 0,C 180,E1 -550.877,E2 -550.877} C_VEL
LIN {X 0,Y 602.488,Z 309.058,A -85,B 0,C 180,E1 -551.599,E2 -551.599} C_VEL
LIN {X 0,Y 601.464,Z 309.183,A -85,B 0,C 180,E1 -552.155,E2 -552.155} C_VEL
LIN {X 0,Y 601.381,Z 309.194,A -85,B 0,C 180,E1 -552.344,E2 -552.344} C_VEL
LIN {X 0,Y 601.392,Z 309.2,A -85,B 0,C 180,E1 -554.898,E2 -554.898} C_VEL
LIN {X 0,Y 601.382,Z 309.194,A -85,B 0,C 180,E1 -557.689,E2 -557.689} C_VEL
LIN {X 0,Y 601.406,Z 309.194,A -85,B 0,C 180,E1 -560.523,E2 -560.523} C_VEL
LIN {X 0,Y 601.406,Z 309.193,A -85,B 0,C 180,E1 -563.411,E2 -563.411} C_VEL
LIN {X 0,Y 601.388,Z 309.196,A -85,B 0,C 180,E1 -566.365,E2 -566.365} C_VEL
LIN {X 0,Y 601.431,Z 309.198,A -85,B 0,C 180,E1 -568.791,E2 -568.791} C_VEL
LIN {X 0,Y 601.401,Z 309.191,A -85,B 0,C 180,E1 -571.727,E2 -571.727} C_VEL
LIN {X 0,Y 601.422,Z 309.19,A -85,B 0,C 180,E1 -574.119,E2 -574.119} C_VEL
LIN {X 0,Y 601.431,Z 309.188,A -85,B 0,C 180,E1 -577.384,E2 -577.384} C_VEL
LIN {X 0,Y 601.403,Z 309.193,A -85,B 0,C 180,E1 -579.996,E2 -579.996} C_VEL
LIN {X 0,Y 601.409,Z 309.198,A -85,B 0,C 180,E1 -582.671,E2 -582.671} C_VEL
LIN {X 0,Y 601.394,Z 309.192,A -85,B 0,C 180,E1 -585.481,E2 -585.481} C_VEL
LIN {X 0,Y 601.421,Z 309.199,A -85,B 0,C 180,E1 -588.408,E2 -588.408} C_VEL
LIN {X 0,Y 601.434,Z 309.189,A -85,B 0,C 180,E1 -590.877,E2 -590.877} C_VEL
LIN {X 0,Y 601.402,Z 309.191,A -85,B 0,C 180,E1 -593.418,E2 -593.418} C_VEL
LIN {X 0,Y 601.432,Z 309.195,A -85,B 0,C 180,E1 -596.065,E2 -596.065} C_VEL
LIN {X 0,Y 601.42,Z 309.193,A -85,B 0,C 180,E1 -598.546,E2 -598.546} C_VEL
LIN {X 0,Y 601.43,Z 309.189,A -85,B 0,C 180,E1 -601.374,E2 -601.374} C_VEL
LIN {X 0,Y 601.452,Z 309.219,A -85,B 0,C 180,E1 -603.171,E2 -603.171} C_VEL
LIN {X 0,Y 601.563,Z 322.417,A -85,B 0,C 180,E1 -605.129,E2 -605.129} C_VEL
LIN {X 0,Y 601.521,Z 342.72,A -85,B 0,C 180,E1 -608.091,E2 -608.091} C_VEL
LIN {X 0,Y 601.812,Z 348.167,A -85,B 0,C 180,E1 -608.169,E2 -608.169} C_VEL
LIN {X 0,Y 601.742,Z 479.738,A -85,B 0,C 180,E1 -609.78,E2 -609.78} C_VEL
LIN {X 0,Y 601.712,Z 493.858,A -85,B 0,C 180,E1 -610.091,E2 -610.091} C_VEL
LIN {X 0,Y 601.666,Z 507.087,A -85,B 0,C 180,E1 -610.511,E2 -610.511} C_VEL
LIN {X 0,Y 601.603,Z 520.48,A -85,B 0,C 180,E1 -611.078,E2 -611.078} C_VEL
LIN {X 0,Y 601.546,Z 533.59,A -85,B 0,C 180,E1 -611.789,E2 -611.789} C_VEL
LIN {X 0,Y 601.516,Z 545.345,A -85,B 0,C 180,E1 -612.579,E2 -612.579} C_VEL
LIN {X 0,Y 601.461,Z 556.329,A -85,B 0,C 180,E1 -613.475,E2 -613.475} C_VEL
LIN {X 0,Y 601.421,Z 565.854,A -85,B 0,C 180,E1 -614.409,E2 -614.409} C_VEL
LIN {X 0,Y 601.403,Z 574.696,A -85,B 0,C 180,E1 -615.449,E2 -615.449} C_VEL
LIN {X 0,Y 601.376,Z 583.094,A -85,B 0,C 180,E1 -616.656,E2 -616.656} C_VEL
LIN {X 0,Y 601.377,Z 589.805,A -85,B 0,C 180,E1 -617.857,E2 -617.857} C_VEL
LIN {X 0,Y 601.348,Z 595.722,A -85,B 0,C 180,E1 -619.223,E2 -619.223} C_VEL
LIN {X 0,Y 601.336,Z 600.02,A -85,B 0,C 180,E1 -620.583,E2 -620.583} C_VEL
LIN {X 0,Y 601.332,Z 602.839,A -85,B 0,C 180,E1 -621.938,E2 -621.938} C_VEL
LIN {X 0,Y 601.349,Z 604.355,A -85,B 0,C 180,E1 -623.417,E2 -623.417} C_VEL
LIN {X 0,Y 601.334,Z 604.368,A -85,B 0,C 180,E1 -624.635,E2 -624.635} C_VEL
LIN {X 0,Y 601.341,Z 603.122,A -85,B 0,C 180,E1 -625.979,E2 -625.979} C_VEL
LIN {X 0,Y 601.318,Z 600.512,A -85,B 0,C 180,E1 -627.32,E2 -627.32} C_VEL
LIN {X 0,Y 601.351,Z 596.481,A -85,B 0,C 180,E1 -628.661,E2 -628.661} C_VEL
LIN {X 0,Y 601.359,Z 590.923,A -85,B 0,C 180,E1 -630,E2 -630} C_VEL
LIN {X 0,Y 601.385,Z 584.666,A -85,B 0,C 180,E1 -631.172,E2 -631.172} C_VEL
LIN {X 0,Y 601.395,Z 576.905,A -85,B 0,C 180,E1 -632.344,E2 -632.344} C_VEL
LIN {X 0,Y 601.397,Z 568.829,A -85,B 0,C 180,E1 -633.35,E2 -633.35} C_VEL
LIN {X 0,Y 601.45,Z 559.134,A -85,B 0,C 180,E1 -634.356,E2 -634.356} C_VEL
LIN {X 0,Y 601.489,Z 548.41,A -85,B 0,C 180,E1 -635.279,E2 -635.279} C_VEL
LIN {X 0,Y 601.566,Z 536.303,A -85,B 0,C 180,E1 -636.135,E2 -636.135} C_VEL
LIN {X 0,Y 601.623,Z 523.226,A -85,B 0,C 180,E1 -636.876,E2 -636.876} C_VEL
LIN {X 0,Y 601.672,Z 510.023,A -85,B 0,C 180,E1 -637.466,E2 -637.466} C_VEL
LIN {X 0,Y 601.691,Z 496.314,A -85,B 0,C 180,E1 -637.93,E2 -637.93} C_VEL
LIN {X 0,Y 601.714,Z 481.998,A -85,B 0,C 180,E1 -638.268,E2 -638.268} C_VEL
LIN {X 0,Y 601.731,Z 460.333,A -85,B 0,C 180,E1 -638.564,E2 -638.564} C_VEL
LIN {X 0,Y 601.673,Z 343.874,A -85,B 0,C 180,E1 -639.976,E2 -639.976} C_VEL
LIN {X 0,Y 601.494,Z 342.66,A -85,B 0,C 180,E1 -640.009,E2 -640.009} C_VEL
LIN {X 0,Y 601.544,Z 323.343,A -85,B 0,C 180,E1 -642.825,E2 -642.825} C_VEL
LIN {X 0,Y 601.471,Z 309.369,A -85,B 0,C 180,E1 -644.895,E2 -644.895} C_VEL
LIN {X 0,Y 601.416,Z 309.19,A -85,B 0,C 180,E1 -646.986,E2 -646.986} C_VEL
LIN {X 0,Y 601.403,Z 309.2,A -85,B 0,C 180,E1 -649.809,E2 -649.809} C_VEL
LIN {X 0,Y 601.415,Z 309.19,A -85,B 0,C 180,E1 -652.682,E2 -652.682} C_VEL
LIN {X 0,Y 601.401,Z 309.191,A -85,B 0,C 180,E1 -654.878,E2 -654.878} C_VEL
LIN {X 0,Y 601.416,Z 309.193,A -85,B 0,C 180,E1 -657.361,E2 -657.361} C_VEL
LIN {X 0,Y 601.422,Z 309.193,A -85,B 0,C 180,E1 -659.392,E2 -659.392} C_VEL
LIN {X 0,Y 601.41,Z 309.2,A -85,B 0,C 180,E1 -661.725,E2 -661.725} C_VEL
LIN {X 0,Y 601.428,Z 309.19,A -85,B 0,C 180,E1 -664.117,E2 -664.117} C_VEL
LIN {X 0,Y 601.401,Z 309.191,A -85,B 0,C 180,E1 -666.582,E2 -666.582} C_VEL
LIN {X 0,Y 601.437,Z 309.197,A -85,B 0,C 180,E1 -669.535,E2 -669.535} C_VEL
LIN {X 0,Y 601.415,Z 309.195,A -85,B 0,C 180,E1 -671.764,E2 -671.764} C_VEL
LIN {X 0,Y 601.42,Z 309.188,A -85,B 0,C 180,E1 -674.534,E2 -674.534} C_VEL
LIN {X 0,Y 601.406,Z 309.2,A -85,B 0,C 180,E1 -677.408,E2 -677.408} C_VEL
LIN {X 0,Y 601.395,Z 309.193,A -85,B 0,C 180,E1 -680.003,E2 -680.003} C_VEL
LIN {X 0,Y 601.43,Z 309.188,A -85,B 0,C 180,E1 -682.616,E2 -682.616} C_VEL
LIN {X 0,Y 601.439,Z 309.194,A -85,B 0,C 180,E1 -685.069,E2 -685.069} C_VEL
LIN {X 0,Y 601.412,Z 309.195,A -85,B 0,C 180,E1 -687.483,E2 -687.483} C_VEL
LIN {X 0,Y 601.39,Z 309.193,A -85,B 0,C 180,E1 -689.855,E2 -689.855} C_VEL
LIN {X 0,Y 601.383,Z 309.193,A -85,B 0,C 180,E1 -692.13,E2 -692.13} C_VEL
LIN {X 0,Y 601.417,Z 309.19,A -85,B 0,C 180,E1 -694.381,E2 -694.381} C_VEL
LIN {X 0,Y 601.397,Z 309.195,A -85,B 0,C 180,E1 -697.395,E2 -697.395} C_VEL
LIN {X 0,Y 601.384,Z 309.193,A -85,B 0,C 180,E1 -700.19,E2 -700.19} C_VEL
LIN {X 0,Y 601.399,Z 309.199,A -85,B 0,C 180,E1 -703.013,E2 -703.013} C_VEL
LIN {X 0,Y 601.39,Z 309.192,A -85,B 0,C 180,E1 -705.794,E2 -705.794} C_VEL
LIN {X 0,Y 601.422,Z 309.194,A -85,B 0,C 180,E1 -708.541,E2 -708.541} C_VEL
LIN {X 0,Y 601.379,Z 309.196,A -85,B 0,C 180,E1 -711.261,E2 -711.261} C_VEL
LIN {X 0,Y 601.374,Z 309.195,A -85,B 0,C 180,E1 -713.378,E2 -713.378} C_VEL
LIN {X 0,Y 601.371,Z 309.195,A -85,B 0,C 180,E1 -715.307,E2 -715.307} C_VEL
LIN {X 0,Y 601.389,Z 309.193,A -85,B 0,C 180,E1 -717.32,E2 -717.32} C_VEL
LIN {X 0,Y 601.4,Z 309.193,A -85,B 0,C 180,E1 -720,E2 -720} C_VEL
LIN {X 0,Y 601.429,Z 309.194,A -85,B 0,C 180,E1 -722.679,E2 -722.679} C_VEL
LIN {X 0,Y 601.366,Z 309.195,A -85,B 0,C 180,E1 -725.364,E2 -725.364} C_VEL
LIN {X 0,Y 601.349,Z 309.197,A -85,B 0,C 180,E1 -727.386,E2 -727.386} C_VEL
LIN {X 0,Y 601.399,Z 309.196,A -85,B 0,C 180,E1 -730.095,E2 -730.095} C_VEL
LIN {X 0,Y 601.392,Z 309.195,A -85,B 0,C 180,E1 -732.829,E2 -732.829} C_VEL
LIN {X 0,Y 601.37,Z 309.196,A -85,B 0,C 180,E1 -735.592,E2 -735.592} C_VEL
LIN {X 0,Y 601.36,Z 309.198,A -85,B 0,C 180,E1 -737.689,E2 -737.689} C_VEL
LIN {X 0,Y 601.418,Z 309.193,A -85,B 0,C 180,E1 -740.522,E2 -740.522} C_VEL
LIN {X 0,Y 601.372,Z 309.195,A -85,B 0,C 180,E1 -743.412,E2 -743.412} C_VEL
LIN {X 0,Y 601.389,Z 309.199,A -85,B 0,C 180,E1 -745.866,E2 -745.866} C_VEL
LIN {X 0,Y 601.412,Z 309.19,A -85,B 0,C 180,E1 -748.788,E2 -748.788} C_VEL
LIN {X 0,Y 601.403,Z 309.193,A -85,B 0,C 180,E1 -751.455,E2 -751.455} C_VEL
LIN {X 0,Y 601.416,Z 309.196,A -85,B 0,C 180,E1 -754.119,E2 -754.119} C_VEL
LIN {X 0,Y 601.389,Z 309.193,A -85,B 0,C 180,E1 -756.584,E2 -756.584} C_VEL
LIN {X 0,Y 601.394,Z 309.193,A -85,B 0,C 180,E1 -759.128,E2 -759.128} C_VEL
LIN {X 0,Y 601.419,Z 309.199,A -85,B 0,C 180,E1 -761.766,E2 -761.766} C_VEL
LIN {X 0,Y 601.417,Z 309.189,A -85,B 0,C 180,E1 -764.536,E2 -764.536} C_VEL
LIN {X 0,Y 601.408,Z 309.196,A -85,B 0,C 180,E1 -767.41,E2 -767.41} C_VEL
LIN {X 0,Y 601.399,Z 309.195,A -85,B 0,C 180,E1 -770.005,E2 -770.005} C_VEL
LIN {X 0,Y 601.427,Z 309.188,A -85,B 0,C 180,E1 -772.619,E2 -772.619} C_VEL
LIN {X 0,Y 601.401,Z 309.195,A -85,B 0,C 180,E1 -775.068,E2 -775.068} C_VEL
LIN {X 0,Y 601.433,Z 309.197,A -85,B 0,C 180,E1 -777.485,E2 -777.485} C_VEL
LIN {X 0,Y 601.427,Z 309.191,A -85,B 0,C 180,E1 -779.852,E2 -779.852} C_VEL
LIN {X 0,Y 601.407,Z 309.191,A -85,B 0,C 180,E1 -782.639,E2 -782.639} C_VEL
LIN {X 0,Y 601.396,Z 309.2,A -85,B 0,C 180,E1 -785.122,E2 -785.122} C_VEL
LIN {X 0,Y 601.44,Z 309.316,A -85,B 0,C 180,E1 -786.18,E2 -786.18} C_VEL
LIN {X 0,Y 601.726,Z 314.049,A -85,B 0,C 180,E1 -786.803,E2 -786.803} C_VEL
LIN {X 0,Y 601.659,Z 335.103,A -85,B 0,C 180,E1 -789.487,E2 -789.487} C_VEL
LIN {X 0,Y 601.576,Z 357.712,A -85,B 0,C 180,E1 -792.318,E2 -792.318} C_VEL
LIN {X 0,Y 601.539,Z 371.577,A -85,B 0,C 180,E1 -794.032,E2 -794.032} C_VEL
LIN {X 0,Y 601.848,Z 377.442,A -85,B 0,C 180,E1 -794.117,E2 -794.117} C_VEL
LIN {X 0,Y 601.753,Z 508.934,A -85,B 0,C 180,E1 -795.721,E2 -795.721} C_VEL
LIN {X 0,Y 601.713,Z 523.294,A -85,B 0,C 180,E1 -796.029,E2 -796.029} C_VEL
LIN {X 0,Y 601.651,Z 537.722,A -85,B 0,C 180,E1 -796.49,E2 -796.49} C_VEL
LIN {X 0,Y 601.609,Z 551.641,A -85,B 0,C 180,E1 -797.09,E2 -797.09} C_VEL
LIN {X 0,Y 601.546,Z 564.099,A -85,B 0,C 180,E1 -797.775,E2 -797.775} C_VEL
LIN {X 0,Y 601.504,Z 575.477,A -85,B 0,C 180,E1 -798.544,E2 -798.544} C_VEL
LIN {X 0,Y 601.482,Z 585.935,A -85,B 0,C 180,E1 -799.396,E2 -799.396} C_VEL
LIN {X 0,Y 601.43,Z 596.337,A -85,B 0,C 180,E1 -800.415,E2 -800.415} C_VEL
LIN {X 0,Y 601.406,Z 604.915,A -85,B 0,C 180,E1 -801.432,E2 -801.432} C_VEL
LIN {X 0,Y 601.392,Z 613.115,A -85,B 0,C 180,E1 -802.615,E2 -802.615} C_VEL
LIN {X 0,Y 601.361,Z 618.751,A -85,B 0,C 180,E1 -803.604,E2 -803.604} C_VEL
LIN {X 0,Y 601.355,Z 623.568,A -85,B 0,C 180,E1 -804.635,E2 -804.635} C_VEL
LIN {X 0,Y 601.343,Z 628.442,A -85,B 0,C 180,E1 -805.979,E2 -805.979} C_VEL
LIN {X 0,Y 601.324,Z 631.831,A -85,B 0,C 180,E1 -807.321,E2 -807.321} C_VEL
LIN {X 0,Y 601.342,Z 633.831,A -85,B 0,C 180,E1 -808.661,E2 -808.661} C_VEL
LIN {X 0,Y 601.333,Z 634.5,A -85,B 0,C 180,E1 -810,E2 -810} C_VEL
LIN {X 0,Y 601.342,Z 633.831,A -85,B 0,C 180,E1 -811.339,E2 -811.339} C_VEL
LIN {X 0,Y 601.324,Z 631.832,A -85,B 0,C 180,E1 -812.68,E2 -812.68} C_VEL
LIN {X 0,Y 601.343,Z 628.442,A -85,B 0,C 180,E1 -814.021,E2 -814.021} C_VEL
LIN {X 0,Y 601.355,Z 623.568,A -85,B 0,C 180,E1 -815.365,E2 -815.365} C_VEL
LIN {X 0,Y 601.355,Z 617.052,A -85,B 0,C 180,E1 -816.711,E2 -816.711} C_VEL
LIN {X 0,Y 601.398,Z 609.799,A -85,B 0,C 180,E1 -817.892,E2 -817.892} C_VEL
LIN {X 0,Y 601.43,Z 600.825,A -85,B 0,C 180,E1 -819.076,E2 -819.076} C_VEL
LIN {X 0,Y 601.44,Z 591.394,A -85,B 0,C 180,E1 -820.095,E2 -820.095} C_VEL
LIN {X 0,Y 601.505,Z 580.695,A -85,B 0,C 180,E1 -821.05,E2 -821.05} C_VEL
LIN {X 0,Y 601.544,Z 569.431,A -85,B 0,C 180,E1 -821.883,E2 -821.883} C_VEL
LIN {X 0,Y 601.565,Z 556.65,A -85,B 0,C 180,E1 -822.653,E2 -822.653} C_VEL
LIN {X 0,Y 601.626,Z 544.167,A -85,B 0,C 180,E1 -823.253,E2 -823.253} C_VEL
LIN {X 0,Y 601.691,Z 530.838,A -85,B 0,C 180,E1 -823.749,E2 -823.749} C_VEL
LIN {X 0,Y 601.733,Z 516.526,A -85,B 0,C 180,E1 -824.134,E2 -824.134} C_VEL
LIN {X 0,Y 601.745,Z 502.124,A -85,B 0,C 180,E1 -824.376,E2 -824.376} C_VEL
LIN {X 0,Y 601.678,Z 372.522,A -85,B 0,C 180,E1 -825.948,E2 -825.948} C_VEL
LIN {X 0,Y 601.55,Z 371.489,A -85,B 0,C 180,E1 -825.979,E2 -825.979} C_VEL
LIN {X 0,Y 601.627,Z 348.119,A -85,B 0,C 180,E1 -828.877,E2 -828.877} C_VEL
LIN {X 0,Y 601.684,Z 326.625,A -85,B 0,C 180,E1 -831.588,E2 -831.588} C_VEL
LIN {X 0,Y 601.733,Z 311.082,A -85,B 0,C 180,E1 -833.579,E2 -833.579} C_VEL
LIN {X 0,Y 601.421,Z 309.193,A -85,B 0,C 180,E1 -833.866,E2 -833.866} C_VEL
LIN {X 0,Y 601.399,Z 309.198,A -85,B 0,C 180,E1 -836.363,E2 -836.363} C_VEL
LIN {X 0,Y 601.436,Z 309.194,A -85,B 0,C 180,E1 -838.789,E2 -838.789} C_VEL
LIN {X 0,Y 601.415,Z 309.19,A -85,B 0,C 180,E1 -841.454,E2 -841.454} C_VEL
LIN {X 0,Y 601.425,Z 309.192,A -85,B 0,C 180,E1 -844.117,E2 -844.117} C_VEL
LIN {X 0,Y 601.4,Z 309.199,A -85,B 0,C 180,E1 -846.582,E2 -846.582} C_VEL
LIN {X 0,Y 601.401,Z 309.192,A -85,B 0,C 180,E1 -849.126,E2 -849.126} C_VEL
LIN {X 0,Y 601.42,Z 309.19,A -85,B 0,C 180,E1 -851.764,E2 -851.764} C_VEL
LIN {X 0,Y 601.417,Z 309.195,A -85,B 0,C 180,E1 -854.534,E2 -854.534} C_VEL
LIN {X 0,Y 601.404,Z 309.191,A -85,B 0,C 180,E1 -857.408,E2 -857.408} C_VEL
LIN {X 0,Y 601.394,Z 309.199,A -85,B 0,C 180,E1 -860.004,E2 -860.004} C_VEL
LIN {X 0,Y 601.419,Z 309.192,A -85,B 0,C 180,E1 -862.618,E2 -862.618} C_VEL
LIN {X 0,Y 601.379,Z 309.193,A -85,B 0,C 180,E1 -865.066,E2 -865.066} C_VEL
LIN {X 0,Y 601.423,Z 309.19,A -85,B 0,C 180,E1 -867.484,E2 -867.484} C_VEL
LIN {X 0,Y 601.417,Z 309.197,A -85,B 0,C 180,E1 -869.851,E2 -869.851} C_VEL
LIN {X 0,Y 601.388,Z 309.2,A -85,B 0,C 180,E1 -872.131,E2 -872.131} C_VEL
LIN {X 0,Y 601.381,Z 309.196,A -85,B 0,C 180,E1 -874.38,E2 -874.38} C_VEL
LIN {X 0,Y 601.368,Z 309.196,A -85,B 0,C 180,E1 -876.588,E2 -876.588} C_VEL
LIN {X 0,Y 601.416,Z 309.194,A -85,B 0,C 180,E1 -879.478,E2 -879.478} C_VEL
LIN {X 0,Y 601.357,Z 309.198,A -85,B 0,C 180,E1 -882.311,E2 -882.311} C_VEL
LIN {X 0,Y 601.368,Z 309.196,A -85,B 0,C 180,E1 -884.408,E2 -884.408} C_VEL
LIN {X 0,Y 601.387,Z 309.196,A -85,B 0,C 180,E1 -887.171,E2 -887.171} C_VEL
LIN {X 0,Y 601.375,Z 309.199,A -85,B 0,C 180,E1 -889.904,E2 -889.904} C_VEL
LIN {X 0,Y 601.348,Z 309.197,A -85,B 0,C 180,E1 -892.614,E2 -892.614} C_VEL
LIN {X 0,Y 601.416,Z 309.197,A -85,B 0,C 180,E1 -895.308,E2 -895.308} C_VEL
LIN {X 0,Y 601.382,Z 309.195,A -85,B 0,C 180,E1 -897.991,E2 -897.991} C_VEL
LIN {X 0,Y 601.402,Z 309.192,A -85,B 0,C 180,E1 -900,E2 -900} C_VEL
LIN {X 0,Y 601.396,Z 309.193,A -85,B 0,C 180,E1 -902.679,E2 -902.679} C_VEL
LIN {X 0,Y 601.425,Z 309.197,A -85,B 0,C 180,E1 -905.364,E2 -905.364} C_VEL
LIN {X 0,Y 601.387,Z 309.193,A -85,B 0,C 180,E1 -908.062,E2 -908.062} C_VEL
LIN {X 0,Y 601.388,Z 309.197,A -85,B 0,C 180,E1 -910.777,E2 -910.777} C_VEL
LIN {X 0,Y 601.381,Z 309.194,A -85,B 0,C 180,E1 -912.344,E2 -912.344} C_VEL
LIN {X 0,Y 600.717,Z 309.284,A -85,B 0,C 180,E1 -912.903,E2 -912.903} C_VEL
LIN {X 0,Y 597.866,Z 309.643,A -85,B 0,C 180,E1 -913.811,E2 -913.811} C_VEL
LIN {X 0,Y 595.456,Z 309.945,A -85,B 0,C 180,E1 -914.541,E2 -914.541} C_VEL
LIN {X 0,Y 594.421,Z 310.07,A -85,B 0,C 180,E1 -915.105,E2 -915.105} C_VEL
LIN {X 0,Y 594.336,Z 310.077,A -85,B 0,C 180,E1 -915.295,E2 -915.295} C_VEL
LIN {X 0,Y 594.331,Z 310.072,A -85,B 0,C 180,E1 -917.906,E2 -917.906} C_VEL
LIN {X 0,Y 594.386,Z 310.072,A -85,B 0,C 180,E1 -920.777,E2 -920.777} C_VEL
LIN {X 0,Y 594.37,Z 310.067,A -85,B 0,C 180,E1 -923.705,E2 -923.705} C_VEL
LIN {X 0,Y 594.376,Z 310.074,A -85,B 0,C 180,E1 -926.7,E2 -926.7} C_VEL
LIN {X 0,Y 594.372,Z 310.073,A -85,B 0,C 180,E1 -928.999,E2 -928.999} C_VEL
LIN {X 0,Y 594.381,Z 310.065,A -85,B 0,C 180,E1 -931.646,E2 -931.646} C_VEL
LIN {X 0,Y 594.391,Z 310.073,A -85,B 0,C 180,E1 -934.58,E2 -934.58} C_VEL
LIN {X 0,Y 594.382,Z 310.065,A -85,B 0,C 180,E1 -937.61,E2 -937.61} C_VEL
LIN {X 0,Y 594.365,Z 310.078,A -85,B 0,C 180,E1 -940.568,E2 -940.568} C_VEL
LIN {X 0,Y 594.376,Z 310.067,A -85,B 0,C 180,E1 -943.299,E2 -943.299} C_VEL
LIN {X 0,Y 594.356,Z 310.075,A -85,B 0,C 180,E1 -946.162,E2 -946.162} C_VEL
LIN {X 0,Y 594.378,Z 310.074,A -85,B 0,C 180,E1 -948.537,E2 -948.537} C_VEL
LIN {X 0,Y 594.385,Z 310.065,A -85,B 0,C 180,E1 -951.296,E2 -951.296} C_VEL
LIN {X 0,Y 594.351,Z 310.072,A -85,B 0,C 180,E1 -953.757,E2 -953.757} C_VEL
LIN {X 0,Y 594.379,Z 310.076,A -85,B 0,C 180,E1 -956.24,E2 -956.24} C_VEL
LIN {X 0,Y 594.371,Z 310.07,A -85,B 0,C 180,E1 -958.651,E2 -958.651} C_VEL
LIN {X 0,Y 594.384,Z 310.066,A -85,B 0,C 180,E1 -961.043,E2 -961.043} C_VEL
LIN {X 0,Y 594.421,Z 310.233,A -85,B 0,C 180,E1 -963.066,E2 -963.066} C_VEL
LIN {X 0,Y 594.603,Z 319.362,A -85,B 0,C 180,E1 -964.443,E2 -964.443} C_VEL
LIN {X 0,Y 594.52,Z 338.179,A -85,B 0,C 180,E1 -967.231,E2 -967.231} C_VEL
LIN {X 0,Y 594.483,Z 342.727,A -85,B 0,C 180,E1 -967.898,E2 -967.898} C_VEL
LIN {X 0,Y 595.008,Z 347.53,A -85,B 0,C 180,E1 -967.975,E2 -967.975} C_VEL
LIN {X 0,Y 594.851,Z 479.301,A -85,B 0,C 180,E1 -969.603,E2 -969.603} C_VEL
LIN {X 0,Y 594.817,Z 493.575,A -85,B 0,C 180,E1 -969.917,E2 -969.917} C_VEL
LIN {X 0,Y 594.753,Z 507.458,A -85,B 0,C 180,E1 -970.365,E2 -970.365} C_VEL
LIN {X 0,Y 594.651,Z 520.977,A -85,B 0,C 180,E1 -970.949,E2 -970.949} C_VEL
LIN {X 0,Y 594.58,Z 533.821,A -85,B 0,C 180,E1 -971.657,E2 -971.657} C_VEL
LIN {X 0,Y 594.529,Z 545.535,A -85,B 0,C 180,E1 -972.456,E2 -972.456} C_VEL
LIN {X 0,Y 594.434,Z 556.647,A -85,B 0,C 180,E1 -973.377,E2 -973.377} C_VEL
LIN {X 0,Y 594.372,Z 566.8,A -85,B 0,C 180,E1 -974.396,E2 -974.396} C_VEL
LIN {X 0,Y 594.348,Z 575.465,A -85,B 0,C 180,E1 -975.447,E2 -975.447} C_VEL
LIN {X 0,Y 594.3,Z 583.69,A -85,B 0,C 180,E1 -976.668,E2 -976.668} C_VEL
LIN {X 0,Y 594.285,Z 589.458,A -85,B 0,C 180,E1 -977.71,E2 -977.71} C_VEL
LIN {X 0,Y 594.256,Z 595.459,A -85,B 0,C 180,E1 -979.093,E2 -979.093} C_VEL
LIN {X 0,Y 594.258,Z 599.833,A -85,B 0,C 180,E1 -980.47,E2 -980.47} C_VEL
LIN {X 0,Y 594.228,Z 602.723,A -85,B 0,C 180,E1 -981.841,E2 -981.841} C_VEL
LIN {X 0,Y 594.272,Z 604.223,A -85,B 0,C 180,E1 -983.208,E2 -983.208} C_VEL
LIN {X 0,Y 594.25,Z 604.385,A -85,B 0,C 180,E1 -984.571,E2 -984.571} C_VEL
LIN {X 0,Y 594.253,Z 603.217,A -85,B 0,C 180,E1 -985.931,E2 -985.931} C_VEL
LIN {X 0,Y 594.22,Z 600.695,A -85,B 0,C 180,E1 -987.288,E2 -987.288} C_VEL
LIN {X 0,Y 594.254,Z 596.741,A -85,B 0,C 180,E1 -988.645,E2 -988.645} C_VEL
LIN {X 0,Y 594.284,Z 591.261,A -85,B 0,C 180,E1 -990,E2 -990} C_VEL
LIN {X 0,Y 594.323,Z 585.088,A -85,B 0,C 180,E1 -991.186,E2 -991.186} C_VEL
LIN {X 0,Y 594.333,Z 577.422,A -85,B 0,C 180,E1 -992.372,E2 -992.372} C_VEL
LIN {X 0,Y 594.374,Z 567.977,A -85,B 0,C 180,E1 -993.559,E2 -993.559} C_VEL
LIN {X 0,Y 594.464,Z 558.115,A -85,B 0,C 180,E1 -994.577,E2 -994.577} C_VEL
LIN {X 0,Y 594.503,Z 547.176,A -85,B 0,C 180,E1 -995.512,E2 -995.512} C_VEL
LIN {X 0,Y 594.585,Z 535.718,A -85,B 0,C 180,E1 -996.316,E2 -996.316} C_VEL
LIN {X 0,Y 594.681,Z 523.465,A -85,B 0,C 180,E1 -997.017,E2 -997.017} C_VEL
LIN {X 0,Y 594.757,Z 510.773,A -85,B 0,C 180,E1 -997.596,E2 -997.596} C_VEL
LIN {X 0,Y 594.815,Z 497.317,A -85,B 0,C 180,E1 -998.065,E2 -998.065} C_VEL
LIN {X 0,Y 594.852,Z 483.501,A -85,B 0,C 180,E1 -998.407,E2 -998.407} C_VEL
LIN {X 0,Y 594.878,Z 466.189,A -85,B 0,C 180,E1 -998.663,E2 -998.663} C_VEL
LIN {X 0,Y 594.988,Z 345.464,A -85,B 0,C 180,E1 -1000.141,E2 -1000.141} C_VEL
LIN {X 0,Y 594.468,Z 342.58,A -85,B 0,C 180,E1 -1000.214,E2 -1000.214} C_VEL
LIN {X 0,Y 594.611,Z 322.681,A -85,B 0,C 180,E1 -1003.151,E2 -1003.151} C_VEL
LIN {X 0,Y 594.575,Z 311.039,A -85,B 0,C 180,E1 -1004.897,E2 -1004.897} C_VEL
LIN {X 0,Y 594.401,Z 310.068,A -85,B 0,C 180,E1 -1005.077,E2 -1005.077} C_VEL
LIN {X 0,Y 594.38,Z 310.076,A -85,B 0,C 180,E1 -1007.904,E2 -1007.904} C_VEL
LIN {X 0,Y 594.379,Z 310.066,A -85,B 0,C 180,E1 -1010.915,E2 -1010.915} C_VEL
LIN {X 0,Y 594.378,Z 310.074,A -85,B 0,C 180,E1 -1013.704,E2 -1013.704} C_VEL
LIN {X 0,Y 594.384,Z 310.065,A -85,B 0,C 180,E1 -1016.699,E2 -1016.699} C_VEL
LIN {X 0,Y 594.382,Z 310.066,A -85,B 0,C 180,E1 -1018.998,E2 -1018.998} C_VEL
LIN {X 0,Y 594.391,Z 310.074,A -85,B 0,C 180,E1 -1021.644,E2 -1021.644} C_VEL
LIN {X 0,Y 594.399,Z 310.063,A -85,B 0,C 180,E1 -1024.578,E2 -1024.578} C_VEL
LIN {X 0,Y 594.386,Z 310.075,A -85,B 0,C 180,E1 -1027.607,E2 -1027.607} C_VEL
LIN {X 0,Y 594.362,Z 310.067,A -85,B 0,C 180,E1 -1030.566,E2 -1030.566} C_VEL
LIN {X 0,Y 594.362,Z 310.075,A -85,B 0,C 180,E1 -1033.298,E2 -1033.298} C_VEL
LIN {X 0,Y 594.363,Z 310.068,A -85,B 0,C 180,E1 -1036.159,E2 -1036.159} C_VEL
LIN {X 0,Y 594.372,Z 310.074,A -85,B 0,C 180,E1 -1039.177,E2 -1039.177} C_VEL
LIN {X 0,Y 594.372,Z 310.067,A -85,B 0,C 180,E1 -1042.058,E2 -1042.058} C_VEL
LIN {X 0,Y 594.354,Z 310.071,A -85,B 0,C 180,E1 -1044.674,E2 -1044.674} C_VEL
LIN {X 0,Y 594.368,Z 310.075,A -85,B 0,C 180,E1 -1047.088,E2 -1047.088} C_VEL
LIN {X 0,Y 594.359,Z 310.071,A -85,B 0,C 180,E1 -1049.674,E2 -1049.674} C_VEL
LIN {X 0,Y 594.364,Z 310.069,A -85,B 0,C 180,E1 -1052.538,E2 -1052.538} C_VEL
LIN {X 0,Y 594.362,Z 310.074,A -85,B 0,C 180,E1 -1054.806,E2 -1054.806} C_VEL
LIN {X 0,Y 594.348,Z 310.075,A -85,B 0,C 180,E1 -1057.265,E2 -1057.265} C_VEL
LIN {X 0,Y 594.351,Z 310.068,A -85,B 0,C 180,E1 -1059.945,E2 -1059.945} C_VEL
LIN {X 0,Y 594.364,Z 310.076,A -85,B 0,C 180,E1 -1062.806,E2 -1062.806} C_VEL
LIN {X 0,Y 594.359,Z 310.068,A -85,B 0,C 180,E1 -1065.832,E2 -1065.832} C_VEL
LIN {X 0,Y 594.377,Z 310.069,A -85,B 0,C 180,E1 -1068.404,E2 -1068.404} C_VEL
LIN {X 0,Y 594.352,Z 310.073,A -85,B 0,C 180,E1 -1071.157,E2 -1071.157} C_VEL
LIN {X 0,Y 594.345,Z 310.071,A -85,B 0,C 180,E1 -1073.341,E2 -1073.341} C_VEL
LIN {X 0,Y 594.346,Z 310.07,A -85,B 0,C 180,E1 -1075.252,E2 -1075.252} C_VEL
LIN {X 0,Y 594.353,Z 310.07,A -85,B 0,C 180,E1 -1077.967,E2 -1077.967} C_VEL
LIN {X 0,Y 594.407,Z 310.07,A -85,B 0,C 180,E1 -1080.677,E2 -1080.677} C_VEL
LIN {X 0,Y 594.293,Z 310.076,A -85,B 0,C 180,E1 -1083.39,E2 -1083.39} C_VEL
LIN {X 0,Y 594.334,Z 310.071,A -85,B 0,C 180,E1 -1085.428,E2 -1085.428} C_VEL
LIN {X 0,Y 594.323,Z 310.073,A -85,B 0,C 180,E1 -1087.474,E2 -1087.474} C_VEL
LIN {X 0,Y 594.36,Z 310.075,A -85,B 0,C 180,E1 -1090.216,E2 -1090.216} C_VEL
LIN {X 0,Y 594.334,Z 310.072,A -85,B 0,C 180,E1 -1092.984,E2 -1092.984} C_VEL
LIN {X 0,Y 594.343,Z 310.07,A -85,B 0,C 180,E1 -1095.079,E2 -1095.079} C_VEL
LIN {X 0,Y 594.353,Z 310.069,A -85,B 0,C 180,E1 -1097.194,E2 -1097.194} C_VEL
LIN {X 0,Y 594.355,Z 310.077,A -85,B 0,C 180,E1 -1100.054,E2 -1100.054} C_VEL
LIN {X 0,Y 594.339,Z 310.071,A -85,B 0,C 180,E1 -1102.968,E2 -1102.968} C_VEL
LIN {X 0,Y 594.342,Z 310.07,A -85,B 0,C 180,E1 -1105.194,E2 -1105.194} C_VEL
LIN {X 0,Y 594.328,Z 310.074,A -85,B 0,C 180,E1 -1107.519,E2 -1107.519} C_VEL
LIN {X 0,Y 594.373,Z 310.071,A -85,B 0,C 180,E1 -1110.329,E2 -1110.329} C_VEL
LIN {X 0,Y 594.365,Z 310.067,A -85,B 0,C 180,E1 -1112.951,E2 -1112.951} C_VEL
LIN {X 0,Y 594.341,Z 310.073,A -85,B 0,C 180,E1 -1115.41,E2 -1115.41} C_VEL
LIN {X 0,Y 594.38,Z 310.074,A -85,B 0,C 180,E1 -1117.941,E2 -1117.941} C_VEL
LIN {X 0,Y 594.361,Z 310.067,A -85,B 0,C 180,E1 -1120.822,E2 -1120.822} C_VEL
LIN {X 0,Y 594.357,Z 310.072,A -85,B 0,C 180,E1 -1123.3,E2 -1123.3} C_VEL
LIN {X 0,Y 594.36,Z 310.071,A -85,B 0,C 180,E1 -1126.161,E2 -1126.161} C_VEL
LIN {X 0,Y 594.371,Z 310.067,A -85,B 0,C 180,E1 -1128.537,E2 -1128.537} C_VEL
LIN {X 0,Y 594.376,Z 310.072,A -85,B 0,C 180,E1 -1131.297,E2 -1131.297} C_VEL
LIN {X 0,Y 594.39,Z 310.071,A -85,B 0,C 180,E1 -1133.759,E2 -1133.759} C_VEL
LIN {X 0,Y 594.374,Z 310.067,A -85,B 0,C 180,E1 -1136.24,E2 -1136.24} C_VEL
LIN {X 0,Y 594.365,Z 310.068,A -85,B 0,C 180,E1 -1138.65,E2 -1138.65} C_VEL
LIN {X 0,Y 594.382,Z 310.07,A -85,B 0,C 180,E1 -1141.043,E2 -1141.043} C_VEL
LIN {X 0,Y 594.385,Z 310.067,A -85,B 0,C 180,E1 -1143.978,E2 -1143.978} C_VEL
LIN {X 0,Y 594.427,Z 310.199,A -85,B 0,C 180,E1 -1145.997,E2 -1145.997} C_VEL
LIN {X 0,Y 594.847,Z 313.908,A -85,B 0,C 180,E1 -1146.501,E2 -1146.501} C_VEL
LIN {X 0,Y 594.769,Z 333.133,A -85,B 0,C 180,E1 -1148.986,E2 -1148.986} C_VEL
LIN {X 0,Y 594.649,Z 356.299,A -85,B 0,C 180,E1 -1151.927,E2 -1151.927} C_VEL
LIN {X 0,Y 594.54,Z 371.577,A -85,B 0,C 180,E1 -1153.839,E2 -1153.839} C_VEL
LIN {X 0,Y 595.027,Z 375.654,A -85,B 0,C 180,E1 -1153.908,E2 -1153.908} C_VEL
LIN {X 0,Y 594.873,Z 509.908,A -85,B 0,C 180,E1 -1155.57,E2 -1155.57} C_VEL
LIN {X 0,Y 594.817,Z 524.145,A -85,B 0,C 180,E1 -1155.889,E2 -1155.889} C_VEL
LIN {X 0,Y 594.74,Z 537.724,A -85,B 0,C 180,E1 -1156.33,E2 -1156.33} C_VEL
LIN {X 0,Y 594.663,Z 551.644,A -85,B 0,C 180,E1 -1156.937,E2 -1156.937} C_VEL
LIN {X 0,Y 594.574,Z 564.101,A -85,B 0,C 180,E1 -1157.629,E2 -1157.629} C_VEL
LIN {X 0,Y 594.523,Z 576.563,A -85,B 0,C 180,E1 -1158.488,E2 -1158.488} C_VEL
LIN {X 0,Y 594.449,Z 587.84,A -85,B 0,C 180,E1 -1159.441,E2 -1159.441} C_VEL
LIN {X 0,Y 594.368,Z 597.853,A -85,B 0,C 180,E1 -1160.472,E2 -1160.472} C_VEL
LIN {X 0,Y 594.323,Z 606.172,A -85,B 0,C 180,E1 -1161.5,E2 -1161.5} C_VEL
LIN {X 0,Y 594.303,Z 614.127,A -85,B 0,C 180,E1 -1162.697,E2 -1162.697} C_VEL
LIN {X 0,Y 594.279,Z 620.528,A -85,B 0,C 180,E1 -1163.89,E2 -1163.89} C_VEL
LIN {X 0,Y 594.237,Z 626.199,A -85,B 0,C 180,E1 -1165.251,E2 -1165.251} C_VEL
LIN {X 0,Y 594.259,Z 630.315,A -85,B 0,C 180,E1 -1166.61,E2 -1166.61} C_VEL
LIN {X 0,Y 594.24,Z 633,A -85,B 0,C 180,E1 -1167.967,E2 -1167.967} C_VEL
LIN {X 0,Y 594.237,Z 634.332,A -85,B 0,C 180,E1 -1169.322,E2 -1169.322} C_VEL
LIN {X 0,Y 594.237,Z 634.332,A -85,B 0,C 180,E1 -1170.678,E2 -1170.678} C_VEL
LIN {X 0,Y 594.24,Z 633,A -85,B 0,C 180,E1 -1172.033,E2 -1172.033} C_VEL
LIN {X 0,Y 594.259,Z 630.316,A -85,B 0,C 180,E1 -1173.39,E2 -1173.39} C_VEL
LIN {X 0,Y 594.237,Z 626.2,A -85,B 0,C 180,E1 -1174.749,E2 -1174.749} C_VEL
LIN {X 0,Y 594.279,Z 620.527,A -85,B 0,C 180,E1 -1176.11,E2 -1176.11} C_VEL
LIN {X 0,Y 594.303,Z 614.127,A -85,B 0,C 180,E1 -1177.303,E2 -1177.303} C_VEL
LIN {X 0,Y 594.323,Z 606.172,A -85,B 0,C 180,E1 -1178.5,E2 -1178.5} C_VEL
LIN {X 0,Y 594.367,Z 597.852,A -85,B 0,C 180,E1 -1179.528,E2 -1179.528} C_VEL
LIN {X 0,Y 594.448,Z 587.839,A -85,B 0,C 180,E1 -1180.559,E2 -1180.559} C_VEL
LIN {X 0,Y 594.523,Z 576.565,A -85,B 0,C 180,E1 -1181.512,E2 -1181.512} C_VEL
LIN {X 0,Y 594.582,Z 564.101,A -85,B 0,C 180,E1 -1182.371,E2 -1182.371} C_VEL
LIN {X 0,Y 594.663,Z 551.644,A -85,B 0,C 180,E1 -1183.063,E2 -1183.063} C_VEL
LIN {X 0,Y 594.74,Z 537.721,A -85,B 0,C 180,E1 -1183.67,E2 -1183.67} C_VEL
LIN {X 0,Y 594.816,Z 524.142,A -85,B 0,C 180,E1 -1184.111,E2 -1184.111} C_VEL
LIN {X 0,Y 594.858,Z 509.905,A -85,B 0,C 180,E1 -1184.431,E2 -1184.431} C_VEL
LIN {X 0,Y 594.95,Z 373.863,A -85,B 0,C 180,E1 -1186.117,E2 -1186.117} C_VEL
LIN {X 0,Y 594.551,Z 371.489,A -85,B 0,C 180,E1 -1186.172,E2 -1186.172} C_VEL
LIN {X 0,Y 594.678,Z 348.109,A -85,B 0,C 180,E1 -1189.108,E2 -1189.108} C_VEL
LIN {X 0,Y 594.791,Z 326.625,A -85,B 0,C 180,E1 -1191.851,E2 -1191.851} C_VEL
LIN {X 0,Y 594.824,Z 312.495,A -85,B 0,C 180,E1 -1193.685,E2 -1193.685} C_VEL
LIN {X 0,Y 594.4,Z 310.07,A -85,B 0,C 180,E1 -1194.027,E2 -1194.027} C_VEL
LIN {X 0,Y 594.378,Z 310.076,A -85,B 0,C 180,E1 -1196.699,E2 -1196.699} C_VEL
LIN {X 0,Y 594.38,Z 310.07,A -85,B 0,C 180,E1 -1198.998,E2 -1198.998} C_VEL
LIN {X 0,Y 594.374,Z 310.067,A -85,B 0,C 180,E1 -1201.642,E2 -1201.642} C_VEL
LIN {X 0,Y 594.374,Z 310.076,A -85,B 0,C 180,E1 -1204.579,E2 -1204.579} C_VEL
LIN {X 0,Y 594.376,Z 310.067,A -85,B 0,C 180,E1 -1207.086,E2 -1207.086} C_VEL
LIN {X 0,Y 594.354,Z 310.07,A -85,B 0,C 180,E1 -1209.772,E2 -1209.772} C_VEL
LIN {X 0,Y 594.365,Z 310.077,A -85,B 0,C 180,E1 -1212.374,E2 -1212.374} C_VEL
LIN {X 0,Y 594.356,Z 310.068,A -85,B 0,C 180,E1 -1215.19,E2 -1215.19} C_VEL
LIN {X 0,Y 594.377,Z 310.075,A -85,B 0,C 180,E1 -1218.151,E2 -1218.151} C_VEL
LIN {X 0,Y 594.365,Z 310.068,A -85,B 0,C 180,E1 -1221.194,E2 -1221.194} C_VEL
LIN {X 0,Y 594.361,Z 310.072,A -85,B 0,C 180,E1 -1223.756,E2 -1223.756} C_VEL
LIN {X 0,Y 594.362,Z 310.075,A -85,B 0,C 180,E1 -1226.238,E2 -1226.238} C_VEL
LIN {X 0,Y 594.352,Z 310.07,A -85,B 0,C 180,E1 -1228.649,E2 -1228.649} C_VEL
LIN {X 0,Y 594.365,Z 310.066,A -85,B 0,C 180,E1 -1231.042,E2 -1231.042} C_VEL
LIN {X 0,Y 594.349,Z 310.077,A -85,B 0,C 180,E1 -1234.055,E2 -1234.055} C_VEL
LIN {X 0,Y 594.36,Z 310.071,A -85,B 0,C 180,E1 -1236.295,E2 -1236.295} C_VEL
LIN {X 0,Y 594.386,Z 310.067,A -85,B 0,C 180,E1 -1239.224,E2 -1239.224} C_VEL
LIN {X 0,Y 594.322,Z 310.077,A -85,B 0,C 180,E1 -1242.094,E2 -1242.094} C_VEL
LIN {X 0,Y 594.33,Z 310.074,A -85,B 0,C 180,E1 -1244.218,E2 -1244.218} C_VEL
LIN {X 0,Y 594.334,Z 310.073,A -85,B 0,C 180,E1 -1246.32,E2 -1246.32} C_VEL
LIN {X 0,Y 594.346,Z 310.072,A -85,B 0,C 180,E1 -1249.094,E2 -1249.094} C_VEL
LIN {X 0,Y 594.333,Z 310.076,A -85,B 0,C 180,E1 -1251.842,E2 -1251.842} C_VEL
LIN {X 0,Y 594.325,Z 310.076,A -85,B 0,C 180,E1 -1253.891,E2 -1253.891} C_VEL
LIN {X 0,Y 594.316,Z 310.076,A -85,B 0,C 180,E1 -1255.932,E2 -1255.932} C_VEL
LIN {X 0,Y 594.356,Z 310.07,A -85,B 0,C 180,E1 -1257.967,E2 -1257.967} C_VEL
LIN {X 0,Y 594.373,Z 310.068,A -85,B 0,C 180,E1 -1260,E2 -1260} C_VEL
LIN {X 0,Y 594.366,Z 310.068,A -85,B 0,C 180,E1 -1262.711,E2 -1262.711} C_VEL
LIN {X 0,Y 594.385,Z 310.072,A -85,B 0,C 180,E1 -1265.428,E2 -1265.428} C_VEL
LIN {X 0,Y 594.339,Z 310.07,A -85,B 0,C 180,E1 -1268.158,E2 -1268.158} C_VEL
LIN {X 0,Y 594.367,Z 310.076,A -85,B 0,C 180,E1 -1271.07,E2 -1271.07} C_VEL
LIN {X 0,Y 594.36,Z 310.07,A -85,B 0,C 180,E1 -1273.68,E2 -1273.68} C_VEL
LIN {X 0,Y 594.336,Z 310.077,A -85,B 0,C 180,E1 -1275.295,E2 -1275.295} C_VEL
LIN {X 0,Y 593.665,Z 310.157,A -85,B 0,C 180,E1 -1275.861,E2 -1275.861} C_VEL
LIN {X 0,Y 590.799,Z 310.517,A -85,B 0,C 180,E1 -1276.779,E2 -1276.779} C_VEL
LIN {X 0,Y 588.387,Z 310.815,A -85,B 0,C 180,E1 -1277.518,E2 -1277.518} C_VEL
LIN {X 0,Y 587.363,Z 310.94,A -85,B 0,C 180,E1 -1278.088,E2 -1278.088} C_VEL
LIN {X 0,Y 587.287,Z 310.95,A -85,B 0,C 180,E1 -1278.281,E2 -1278.281} C_VEL
LIN {X 0,Y 587.319,Z 310.954,A -85,B 0,C 180,E1 -1281.038,E2 -1281.038} C_VEL
LIN {X 0,Y 587.308,Z 310.951,A -85,B 0,C 180,E1 -1283.26,E2 -1283.26} C_VEL
LIN {X 0,Y 587.321,Z 310.946,A -85,B 0,C 180,E1 -1285.518,E2 -1285.518} C_VEL
LIN {X 0,Y 587.336,Z 310.943,A -85,B 0,C 180,E1 -1287.819,E2 -1287.819} C_VEL
LIN {X 0,Y 587.323,Z 310.951,A -85,B 0,C 180,E1 -1290.51,E2 -1290.51} C_VEL
LIN {X 0,Y 587.331,Z 310.947,A -85,B 0,C 180,E1 -1293.113,E2 -1293.113} C_VEL
LIN {X 0,Y 587.294,Z 310.948,A -85,B 0,C 180,E1 -1295.539,E2 -1295.539} C_VEL
LIN {X 0,Y 587.331,Z 310.944,A -85,B 0,C 180,E1 -1297.839,E2 -1297.839} C_VEL
LIN {X 0,Y 587.312,Z 310.951,A -85,B 0,C 180,E1 -1300.255,E2 -1300.255} C_VEL
LIN {X 0,Y 587.321,Z 310.947,A -85,B 0,C 180,E1 -1303.121,E2 -1303.121} C_VEL
LIN {X 0,Y 587.308,Z 310.951,A -85,B 0,C 180,E1 -1306.05,E2 -1306.05} C_VEL
LIN {X 0,Y 587.334,Z 310.946,A -85,B 0,C 180,E1 -1308.926,E2 -1308.926} C_VEL
LIN {X 0,Y 587.33,Z 310.945,A -85,B 0,C 180,E1 -1311.522,E2 -1311.522} C_VEL
LIN {X 0,Y 587.345,Z 310.949,A -85,B 0,C 180,E1 -1314.457,E2 -1314.457} C_VEL
LIN {X 0,Y 587.339,Z 310.945,A -85,B 0,C 180,E1 -1316.889,E2 -1316.889} C_VEL
LIN {X 0,Y 587.335,Z 310.949,A -85,B 0,C 180,E1 -1319.831,E2 -1319.831} C_VEL
LIN {X 0,Y 587.408,Z 311.092,A -85,B 0,C 180,E1 -1322.935,E2 -1322.935} C_VEL
LIN {X 0,Y 587.654,Z 317.034,A -85,B 0,C 180,E1 -1323.849,E2 -1323.849} C_VEL
LIN {X 0,Y 587.549,Z 335.095,A -85,B 0,C 180,E1 -1326.565,E2 -1326.565} C_VEL
LIN {X 0,Y 587.465,Z 342.734,A -85,B 0,C 180,E1 -1327.7,E2 -1327.7} C_VEL
LIN {X 0,Y 588.19,Z 346.875,A -85,B 0,C 180,E1 -1327.776,E2 -1327.776} C_VEL
LIN {X 0,Y 587.975,Z 478.823,A -85,B 0,C 180,E1 -1329.422,E2 -1329.422} C_VEL
LIN {X 0,Y 587.92,Z 493.289,A -85,B 0,C 180,E1 -1329.74,E2 -1329.74} C_VEL
LIN {X 0,Y 587.84,Z 507.827,A -85,B 0,C 180,E1 -1330.215,E2 -1330.215} C_VEL
LIN {X 0,Y 587.732,Z 520.863,A -85,B 0,C 180,E1 -1330.786,E2 -1330.786} C_VEL
LIN {X 0,Y 587.621,Z 534.053,A -85,B 0,C 180,E1 -1331.522,E2 -1331.522} C_VEL
LIN {X 0,Y 587.542,Z 545.725,A -85,B 0,C 180,E1 -1332.331,E2 -1332.331} C_VEL
LIN {X 0,Y 587.402,Z 557.372,A -85,B 0,C 180,E1 -1333.313,E2 -1333.313} C_VEL
LIN {X 0,Y 587.336,Z 567.685,A -85,B 0,C 180,E1 -1334.382,E2 -1334.382} C_VEL
LIN {X 0,Y 587.289,Z 576.197,A -85,B 0,C 180,E1 -1335.446,E2 -1335.446} C_VEL
LIN {X 0,Y 587.248,Z 584.289,A -85,B 0,C 180,E1 -1336.681,E2 -1336.681} C_VEL
LIN {X 0,Y 587.205,Z 590.756,A -85,B 0,C 180,E1 -1337.91,E2 -1337.91} C_VEL
LIN {X 0,Y 587.189,Z 596.451,A -85,B 0,C 180,E1 -1339.309,E2 -1339.309} C_VEL
LIN {X 0,Y 587.157,Z 599.645,A -85,B 0,C 180,E1 -1340.354,E2 -1340.354} C_VEL
LIN {X 0,Y 587.138,Z 602.608,A -85,B 0,C 180,E1 -1341.742,E2 -1341.742} C_VEL
LIN {X 0,Y 587.167,Z 604.174,A -85,B 0,C 180,E1 -1343.126,E2 -1343.126} C_VEL
LIN {X 0,Y 587.168,Z 604.402,A -85,B 0,C 180,E1 -1344.505,E2 -1344.505} C_VEL
LIN {X 0,Y 587.168,Z 603.3,A -85,B 0,C 180,E1 -1345.882,E2 -1345.882} C_VEL
LIN {X 0,Y 587.126,Z 600.855,A -85,B 0,C 180,E1 -1347.256,E2 -1347.256} C_VEL
LIN {X 0,Y 587.158,Z 596.997,A -85,B 0,C 180,E1 -1348.628,E2 -1348.628} C_VEL
LIN {X 0,Y 587.192,Z 591.598,A -85,B 0,C 180,E1 -1350,E2 -1350} C_VEL
LIN {X 0,Y 587.258,Z 586.473,A -85,B 0,C 180,E1 -1351.029,E2 -1351.029} C_VEL
LIN {X 0,Y 587.257,Z 579.146,A -85,B 0,C 180,E1 -1352.229,E2 -1352.229} C_VEL
LIN {X 0,Y 587.278,Z 570.072,A -85,B 0,C 180,E1 -1353.43,E2 -1353.43} C_VEL
LIN {X 0,Y 587.371,Z 560.615,A -85,B 0,C 180,E1 -1354.46,E2 -1354.46} C_VEL
LIN {X 0,Y 587.506,Z 549.127,A -85,B 0,C 180,E1 -1355.491,E2 -1355.491} C_VEL
LIN {X 0,Y 587.621,Z 538.333,A -85,B 0,C 180,E1 -1356.289,E2 -1356.289} C_VEL
LIN {X 0,Y 587.672,Z 527.238,A -85,B 0,C 180,E1 -1356.97,E2 -1356.97} C_VEL
LIN {X 0,Y 587.798,Z 513.531,A -85,B 0,C 180,E1 -1357.644,E2 -1357.644} C_VEL
LIN {X 0,Y 587.917,Z 499.705,A -85,B 0,C 180,E1 -1358.161,E2 -1358.161} C_VEL
LIN {X 0,Y 588.008,Z 486.04,A -85,B 0,C 180,E1 -1358.527,E2 -1358.527} C_VEL
LIN {X 0,Y 587.997,Z 472.071,A -85,B 0,C 180,E1 -1358.765,E2 -1358.765} C_VEL
LIN {X 0,Y 588.135,Z 346.112,A -85,B 0,C 180,E1 -1360.325,E2 -1360.325} C_VEL
LIN {X 0,Y 587.475,Z 342.645,A -85,B 0,C 180,E1 -1360.402,E2 -1360.402} C_VEL
LIN {X 0,Y 587.631,Z 323.19,A -85,B 0,C 180,E1 -1363.31,E2 -1363.31} C_VEL
LIN {X 0,Y 587.656,Z 312.709,A -85,B 0,C 180,E1 -1364.899,E2 -1364.899} C_VEL
LIN {X 0,Y 587.362,Z 310.946,A -85,B 0,C 180,E1 -1365.217,E2 -1365.217} C_VEL
LIN {X 0,Y 587.327,Z 310.953,A -85,B 0,C 180,E1 -1368.126,E2 -1368.126} C_VEL
LIN {X 0,Y 587.335,Z 310.944,A -85,B 0,C 180,E1 -1371.037,E2 -1371.037} C_VEL
LIN {X 0,Y 587.317,Z 310.947,A -85,B 0,C 180,E1 -1373.258,E2 -1373.258} C_VEL
LIN {X 0,Y 587.336,Z 310.949,A -85,B 0,C 180,E1 -1375.516,E2 -1375.516} C_VEL
LIN {X 0,Y 587.347,Z 310.951,A -85,B 0,C 180,E1 -1377.817,E2 -1377.817} C_VEL
LIN {X 0,Y 587.333,Z 310.944,A -85,B 0,C 180,E1 -1380.508,E2 -1380.508} C_VEL
LIN {X 0,Y 587.338,Z 310.945,A -85,B 0,C 180,E1 -1383.111,E2 -1383.111} C_VEL
LIN {X 0,Y 587.345,Z 310.951,A -85,B 0,C 180,E1 -1385.543,E2 -1385.543} C_VEL
LIN {X 0,Y 587.328,Z 310.944,A -85,B 0,C 180,E1 -1388.478,E2 -1388.478} C_VEL
LIN {X 0,Y 587.334,Z 310.946,A -85,B 0,C 180,E1 -1391.156,E2 -1391.156} C_VEL
LIN {X 0,Y 587.307,Z 310.948,A -85,B 0,C 180,E1 -1394.111,E2 -1394.111} C_VEL
LIN {X 0,Y 587.31,Z 310.95,A -85,B 0,C 180,E1 -1396.993,E2 -1396.993} C_VEL
LIN {X 0,Y 587.305,Z 310.951,A -85,B 0,C 180,E1 -1399.744,E2 -1399.744} C_VEL
LIN {X 0,Y 587.336,Z 310.943,A -85,B 0,C 180,E1 -1402.391,E2 -1402.391} C_VEL
LIN {X 0,Y 587.341,Z 310.945,A -85,B 0,C 180,E1 -1405.651,E2 -1405.651} C_VEL
LIN {X 0,Y 587.339,Z 310.943,A -85,B 0,C 180,E1 -1408.231,E2 -1408.231} C_VEL
LIN {X 0,Y 587.337,Z 310.949,A -85,B 0,C 180,E1 -1410.866,E2 -1410.866} C_VEL
LIN {X 0,Y 587.325,Z 310.945,A -85,B 0,C 180,E1 -1413.72,E2 -1413.72} C_VEL
LIN {X 0,Y 587.292,Z 310.949,A -85,B 0,C 180,E1 -1415.991,E2 -1415.991} C_VEL
LIN {X 0,Y 587.319,Z 310.954,A -85,B 0,C 180,E1 -1418.962,E2 -1418.962} C_VEL
LIN {X 0,Y 587.328,Z 310.95,A -85,B 0,C 180,E1 -1421.15,E2 -1421.15} C_VEL
LIN {X 0,Y 587.297,Z 310.948,A -85,B 0,C 180,E1 -1424.024,E2 -1424.024} C_VEL
LIN {X 0,Y 587.335,Z 310.944,A -85,B 0,C 180,E1 -1426.153,E2 -1426.153} C_VEL
LIN {X 0,Y 587.322,Z 310.951,A -85,B 0,C 180,E1 -1428.962,E2 -1428.962} C_VEL
LIN {X 0,Y 587.302,Z 310.947,A -85,B 0,C 180,E1 -1431.744,E2 -1431.744} C_VEL
LIN {X 0,Y 587.34,Z 310.949,A -85,B 0,C 180,E1 -1434.507,E2 -1434.507} C_VEL
LIN {X 0,Y 587.33,Z 310.945,A -85,B 0,C 180,E1 -1437.256,E2 -1437.256} C_VEL
LIN {X 0,Y 587.342,Z 310.944,A -85,B 0,C 180,E1 -1440,E2 -1440} C_VEL
LIN {X 0,Y 587.352,Z 310.946,A -85,B 0,C 180,E1 -1442.743,E2 -1442.743} C_VEL
LIN {X 0,Y 587.303,Z 310.947,A -85,B 0,C 180,E1 -1445.493,E2 -1445.493} C_VEL
LIN {X 0,Y 587.286,Z 310.949,A -85,B 0,C 180,E1 -1447.564,E2 -1447.564} C_VEL
LIN {X 0,Y 587.309,Z 310.956,A -85,B 0,C 180,E1 -1450.34,E2 -1450.34} C_VEL
LIN {X 0,Y 587.283,Z 310.95,A -85,B 0,C 180,E1 -1453.142,E2 -1453.142} C_VEL
LIN {X 0,Y 587.301,Z 310.947,A -85,B 0,C 180,E1 -1455.264,E2 -1455.264} C_VEL
LIN {X 0,Y 587.29,Z 310.949,A -85,B 0,C 180,E1 -1457.408,E2 -1457.408} C_VEL
LIN {X 0,Y 587.293,Z 310.95,A -85,B 0,C 180,E1 -1459.577,E2 -1459.577} C_VEL
LIN {X 0,Y 587.301,Z 310.951,A -85,B 0,C 180,E1 -1461.775,E2 -1461.775} C_VEL
LIN {X 0,Y 587.332,Z 310.944,A -85,B 0,C 180,E1 -1464.759,E2 -1464.759} C_VEL
LIN {X 0,Y 587.288,Z 310.949,A -85,B 0,C 180,E1 -1467.048,E2 -1467.048} C_VEL
LIN {X 0,Y 587.329,Z 310.945,A -85,B 0,C 180,E1 -1469.38,E2 -1469.38} C_VEL
LIN {X 0,Y 587.333,Z 310.952,A -85,B 0,C 180,E1 -1471.836,E2 -1471.836} C_VEL
LIN {X 0,Y 587.333,Z 310.947,A -85,B 0,C 180,E1 -1474.348,E2 -1474.348} C_VEL
LIN {X 0,Y 587.338,Z 310.943,A -85,B 0,C 180,E1 -1476.748,E2 -1476.748} C_VEL
LIN {X 0,Y 587.322,Z 310.948,A -85,B 0,C 180,E1 -1479.361,E2 -1479.361} C_VEL
LIN {X 0,Y 587.326,Z 310.948,A -85,B 0,C 180,E1 -1482.109,E2 -1482.109} C_VEL
LIN {X 0,Y 587.308,Z 310.948,A -85,B 0,C 180,E1 -1485.09,E2 -1485.09} C_VEL
LIN {X 0,Y 587.347,Z 310.947,A -85,B 0,C 180,E1 -1487.928,E2 -1487.928} C_VEL
LIN {X 0,Y 587.317,Z 310.949,A -85,B 0,C 180,E1 -1491.06,E2 -1491.06} C_VEL
LIN {X 0,Y 587.348,Z 310.949,A -85,B 0,C 180,E1 -1493.293,E2 -1493.293} C_VEL
LIN {X 0,Y 587.358,Z 310.946,A -85,B 0,C 180,E1 -1495.781,E2 -1495.781} C_VEL
LIN {X 0,Y 587.339,Z 310.944,A -85,B 0,C 180,E1 -1498.232,E2 -1498.232} C_VEL
LIN {X 0,Y 587.348,Z 310.945,A -85,B 0,C 180,E1 -1500.867,E2 -1500.867} C_VEL
LIN {X 0,Y 587.358,Z 310.945,A -85,B 0,C 180,E1 -1503.82,E2 -1503.82} C_VEL
LIN {X 0,Y 587.378,Z 311.089,A -85,B 0,C 180,E1 -1505.809,E2 -1505.809} C_VEL
LIN {X 0,Y 587.999,Z 315.321,A -85,B 0,C 180,E1 -1506.397,E2 -1506.397} C_VEL
LIN {X 0,Y 587.84,Z 335.103,A -85,B 0,C 180,E1 -1508.982,E2 -1508.982} C_VEL
LIN {X 0,Y 587.701,Z 357.712,A -85,B 0,C 180,E1 -1511.886,E2 -1511.886} C_VEL
LIN {X 0,Y 587.563,Z 371.577,A -85,B 0,C 180,E1 -1513.642,E2 -1513.642} C_VEL
LIN {X 0,Y 588.199,Z 375.654,A -85,B 0,C 180,E1 -1513.716,E2 -1513.716} C_VEL
LIN {X 0,Y 588.009,Z 509.907,A -85,B 0,C 180,E1 -1515.398,E2 -1515.398} C_VEL
LIN {X 0,Y 587.935,Z 524.097,A -85,B 0,C 180,E1 -1515.719,E2 -1515.719} C_VEL
LIN {X 0,Y 587.824,Z 537.723,A -85,B 0,C 180,E1 -1516.166,E2 -1516.166} C_VEL
LIN {X 0,Y 587.727,Z 551.646,A -85,B 0,C 180,E1 -1516.78,E2 -1516.78} C_VEL
LIN {X 0,Y 587.608,Z 564.103,A -85,B 0,C 180,E1 -1517.48,E2 -1517.48} C_VEL
LIN {X 0,Y 587.513,Z 576.643,A -85,B 0,C 180,E1 -1518.354,E2 -1518.354} C_VEL
LIN {X 0,Y 587.444,Z 587.839,A -85,B 0,C 180,E1 -1519.314,E2 -1519.314} C_VEL
LIN {X 0,Y 587.319,Z 597.853,A -85,B 0,C 180,E1 -1520.356,E2 -1520.356} C_VEL
LIN {X 0,Y 587.277,Z 606.173,A -85,B 0,C 180,E1 -1521.397,E2 -1521.397} C_VEL
LIN {X 0,Y 587.244,Z 614.127,A -85,B 0,C 180,E1 -1522.608,E2 -1522.608} C_VEL
LIN {X 0,Y 587.203,Z 620.528,A -85,B 0,C 180,E1 -1523.816,E2 -1523.816} C_VEL
LIN {X 0,Y 587.16,Z 624.962,A -85,B 0,C 180,E1 -1524.85,E2 -1524.85} C_VEL
LIN {X 0,Y 587.179,Z 628.443,A -85,B 0,C 180,E1 -1525.882,E2 -1525.882} C_VEL
LIN {X 0,Y 587.13,Z 631.832,A -85,B 0,C 180,E1 -1527.256,E2 -1527.256} C_VEL
LIN {X 0,Y 587.141,Z 633.832,A -85,B 0,C 180,E1 -1528.628,E2 -1528.628} C_VEL
LIN {X 0,Y 587.135,Z 634.5,A -85,B 0,C 180,E1 -1530,E2 -1530} C_VEL
LIN {X 0,Y 587.141,Z 633.832,A -85,B 0,C 180,E1 -1531.372,E2 -1531.372} C_VEL
LIN {X 0,Y 587.13,Z 631.833,A -85,B 0,C 180,E1 -1532.744,E2 -1532.744} C_VEL
LIN {X 0,Y 587.179,Z 628.444,A -85,B 0,C 180,E1 -1534.118,E2 -1534.118} C_VEL
LIN {X 0,Y 587.199,Z 623.568,A -85,B 0,C 180,E1 -1535.494,E2 -1535.494} C_VEL
LIN {X 0,Y 587.209,Z 617.053,A -85,B 0,C 180,E1 -1536.874,E2 -1536.874} C_VEL
LIN {X 0,Y 587.268,Z 609.801,A -85,B 0,C 180,E1 -1538.083,E2 -1538.083} C_VEL
LIN {X 0,Y 587.321,Z 600.825,A -85,B 0,C 180,E1 -1539.296,E2 -1539.296} C_VEL
LIN {X 0,Y 587.372,Z 591.394,A -85,B 0,C 180,E1 -1540.339,E2 -1540.339} C_VEL
LIN {X 0,Y 587.474,Z 581.029,A -85,B 0,C 180,E1 -1541.29,E2 -1541.29} C_VEL
LIN {X 0,Y 587.575,Z 569.435,A -85,B 0,C 180,E1 -1542.17,E2 -1542.17} C_VEL
LIN {X 0,Y 587.668,Z 556.654,A -85,B 0,C 180,E1 -1542.957,E2 -1542.957} C_VEL
LIN {X 0,Y 587.78,Z 544.168,A -85,B 0,C 180,E1 -1543.571,E2 -1543.571} C_VEL
LIN {X 0,Y 587.889,Z 530.617,A -85,B 0,C 180,E1 -1544.085,E2 -1544.085} C_VEL
LIN {X 0,Y 587.946,Z 516.971,A -85,B 0,C 180,E1 -1544.461,E2 -1544.461} C_VEL
LIN {X 0,Y 588.01,Z 502.632,A -85,B 0,C 180,E1 -1544.713,E2 -1544.713} C_VEL
LIN {X 0,Y 588.057,Z 374.309,A -85,B 0,C 180,E1 -1546.305,E2 -1546.305} C_VEL
LIN {X 0,Y 587.582,Z 371.489,A -85,B 0,C 180,E1 -1546.369,E2 -1546.369} C_VEL
LIN {X 0,Y 587.727,Z 349.626,A -85,B 0,C 180,E1 -1549.148,E2 -1549.148} C_VEL
LIN {X 0,Y 587.883,Z 329.451,A -85,B 0,C 180,E1 -1551.752,E2 -1551.752} C_VEL
LIN {X 0,Y 587.916,Z 313.908,A -85,B 0,C 180,E1 -1553.793,E2 -1553.793} C_VEL
LIN {X 0,Y 587.366,Z 310.947,A -85,B 0,C 180,E1 -1554.212,E2 -1554.212} C_VEL
LIN {X 0,Y 587.326,Z 310.949,A -85,B 0,C 180,E1 -1557.046,E2 -1557.046} C_VEL
LIN {X 0,Y 587.346,Z 310.943,A -85,B 0,C 180,E1 -1559.379,E2 -1559.379} C_VEL
LIN {X 0,Y 587.342,Z 310.944,A -85,B 0,C 180,E1 -1561.835,E2 -1561.835} C_VEL
LIN {X 0,Y 587.344,Z 310.95,A -85,B 0,C 180,E1 -1564.347,E2 -1564.347} C_VEL
LIN {X 0,Y 587.347,Z 310.946,A -85,B 0,C 180,E1 -1566.746,E2 -1566.746} C_VEL
LIN {X 0,Y 587.327,Z 310.944,A -85,B 0,C 180,E1 -1569.36,E2 -1569.36} C_VEL
LIN {X 0,Y 587.328,Z 310.95,A -85,B 0,C 180,E1 -1572.107,E2 -1572.107} C_VEL
LIN {X 0,Y 587.309,Z 310.946,A -85,B 0,C 180,E1 -1575.088,E2 -1575.088} C_VEL
LIN {X 0,Y 587.345,Z 310.947,A -85,B 0,C 180,E1 -1577.927,E2 -1577.927} C_VEL
LIN {X 0,Y 587.311,Z 310.947,A -85,B 0,C 180,E1 -1581.059,E2 -1581.059} C_VEL
LIN {X 0,Y 587.339,Z 310.943,A -85,B 0,C 180,E1 -1583.292,E2 -1583.292} C_VEL
LIN {X 0,Y 587.346,Z 310.947,A -85,B 0,C 180,E1 -1585.779,E2 -1585.779} C_VEL
LIN {X 0,Y 587.329,Z 310.949,A -85,B 0,C 180,E1 -1588.23,E2 -1588.23} C_VEL
LIN {X 0,Y 587.332,Z 310.942,A -85,B 0,C 180,E1 -1590.867,E2 -1590.867} C_VEL
LIN {X 0,Y 587.321,Z 310.954,A -85,B 0,C 180,E1 -1593.823,E2 -1593.823} C_VEL
LIN {X 0,Y 587.315,Z 310.954,A -85,B 0,C 180,E1 -1595.993,E2 -1595.993} C_VEL
LIN {X 0,Y 587.299,Z 310.951,A -85,B 0,C 180,E1 -1598.225,E2 -1598.225} C_VEL
LIN {X 0,Y 587.328,Z 310.946,A -85,B 0,C 180,E1 -1601.151,E2 -1601.151} C_VEL
LIN {X 0,Y 587.29,Z 310.953,A -85,B 0,C 180,E1 -1604.024,E2 -1604.024} C_VEL
LIN {X 0,Y 587.319,Z 310.948,A -85,B 0,C 180,E1 -1606.153,E2 -1606.153} C_VEL
LIN {X 0,Y 587.274,Z 310.952,A -85,B 0,C 180,E1 -1608.961,E2 -1608.961} C_VEL
LIN {X 0,Y 587.3,Z 310.954,A -85,B 0,C 180,E1 -1611.744,E2 -1611.744} C_VEL
LIN {X 0,Y 587.284,Z 310.954,A -85,B 0,C 180,E1 -1613.817,E2 -1613.817} C_VEL
LIN {X 0,Y 587.274,Z 310.954,A -85,B 0,C 180,E1 -1615.883,E2 -1615.883} C_VEL
LIN {X 0,Y 587.33,Z 310.946,A -85,B 0,C 180,E1 -1617.943,E2 -1617.943} C_VEL
LIN {X 0,Y 587.344,Z 310.944,A -85,B 0,C 180,E1 -1620,E2 -1620} C_VEL
LIN {X 0,Y 587.336,Z 310.944,A -85,B 0,C 180,E1 -1622.744,E2 -1622.744} C_VEL
LIN {X 0,Y 587.346,Z 310.948,A -85,B 0,C 180,E1 -1625.493,E2 -1625.493} C_VEL
LIN {X 0,Y 587.306,Z 310.946,A -85,B 0,C 180,E1 -1628.256,E2 -1628.256} C_VEL
LIN {X 0,Y 587.335,Z 310.953,A -85,B 0,C 180,E1 -1631.134,E2 -1631.134} C_VEL
LIN {X 0,Y 587.317,Z 310.946,A -85,B 0,C 180,E1 -1634.248,E2 -1634.248} C_VEL
LIN {X 0,Y 587.333,Z 310.95,A -85,B 0,C 180,E1 -1636.814,E2 -1636.814} C_VEL
LIN {X 0,Y 587.287,Z 310.95,A -85,B 0,C 180,E1 -1638.281,E2 -1638.281} C_VEL
LIN {X 0,Y 586.649,Z 311.037,A -85,B 0,C 180,E1 -1638.853,E2 -1638.853} C_VEL
LIN {X 0,Y 583.837,Z 311.39,A -85,B 0,C 180,E1 -1639.782,E2 -1639.782} C_VEL
LIN {X 0,Y 581.431,Z 311.69,A -85,B 0,C 180,E1 -1640.529,E2 -1640.529} C_VEL
LIN {X 0,Y 580.372,Z 311.818,A -85,B 0,C 180,E1 -1641.105,E2 -1641.105} C_VEL
LIN {X 0,Y 580.273,Z 311.827,A -85,B 0,C 180,E1 -1641.301,E2 -1641.301} C_VEL
LIN {X 0,Y 580.262,Z 311.825,A -85,B 0,C 180,E1 -1643.559,E2 -1643.559} C_VEL
LIN {X 0,Y 580.279,Z 311.822,A -85,B 0,C 180,E1 -1645.85,E2 -1645.85} C_VEL
LIN {X 0,Y 580.289,Z 311.822,A -85,B 0,C 180,E1 -1648.187,E2 -1648.187} C_VEL
LIN {X 0,Y 580.277,Z 311.832,A -85,B 0,C 180,E1 -1650.696,E2 -1650.696} C_VEL
LIN {X 0,Y 580.295,Z 311.822,A -85,B 0,C 180,E1 -1653.317,E2 -1653.317} C_VEL
LIN {X 0,Y 580.241,Z 311.827,A -85,B 0,C 180,E1 -1655.758,E2 -1655.758} C_VEL
LIN {X 0,Y 580.281,Z 311.825,A -85,B 0,C 180,E1 -1658.147,E2 -1658.147} C_VEL
LIN {X 0,Y 580.295,Z 311.826,A -85,B 0,C 180,E1 -1660.844,E2 -1660.844} C_VEL
LIN {X 0,Y 580.284,Z 311.822,A -85,B 0,C 180,E1 -1663.658,E2 -1663.658} C_VEL
LIN {X 0,Y 580.27,Z 311.831,A -85,B 0,C 180,E1 -1666.611,E2 -1666.611} C_VEL
LIN {X 0,Y 580.297,Z 311.821,A -85,B 0,C 180,E1 -1669.158,E2 -1669.158} C_VEL
LIN {X 0,Y 580.288,Z 311.826,A -85,B 0,C 180,E1 -1671.928,E2 -1671.928} C_VEL
LIN {X 0,Y 580.299,Z 311.826,A -85,B 0,C 180,E1 -1674.457,E2 -1674.457} C_VEL
LIN {X 0,Y 580.29,Z 311.822,A -85,B 0,C 180,E1 -1676.976,E2 -1676.976} C_VEL
LIN {X 0,Y 580.297,Z 311.822,A -85,B 0,C 180,E1 -1679.426,E2 -1679.426} C_VEL
LIN {X 0,Y 580.301,Z 311.83,A -85,B 0,C 180,E1 -1682.142,E2 -1682.142} C_VEL
LIN {X 0,Y 580.342,Z 311.944,A -85,B 0,C 180,E1 -1682.797,E2 -1682.797} C_VEL
LIN {X 0,Y 580.733,Z 316.918,A -85,B 0,C 180,E1 -1683.58,E2 -1683.58} C_VEL
LIN {X 0,Y 580.568,Z 335.804,A -85,B 0,C 180,E1 -1686.455,E2 -1686.455} C_VEL
LIN {X 0,Y 580.468,Z 342.664,A -85,B 0,C 180,E1 -1687.487,E2 -1687.487} C_VEL
LIN {X 0,Y 581.4,Z 348.094,A -85,B 0,C 180,E1 -1687.596,E2 -1687.596} C_VEL
LIN {X 0,Y 581.112,Z 479.658,A -85,B 0,C 180,E1 -1689.261,E2 -1689.261} C_VEL
LIN {X 0,Y 581.039,Z 493.794,A -85,B 0,C 180,E1 -1689.582,E2 -1689.582} C_VEL
LIN {X 0,Y 580.93,Z 507.029,A -85,B 0,C 180,E1 -1690.016,E2 -1690.016} C_VEL
LIN {X 0,Y 580.819,Z 520.666,A -85,B 0,C 180,E1 -1690.615,E2 -1690.615} C_VEL
LIN {X 0,Y 580.692,Z 532.834,A -85,B 0,C 180,E1 -1691.294,E2 -1691.294} C_VEL
LIN {X 0,Y 580.561,Z 544.721,A -85,B 0,C 180,E1 -1692.111,E2 -1692.111} C_VEL
LIN {X 0,Y 580.421,Z 555.961,A -85,B 0,C 180,E1 -1693.053,E2 -1693.053} C_VEL
LIN {X 0,Y 580.298,Z 565.411,A -85,B 0,C 180,E1 -1694.007,E2 -1694.007} C_VEL
LIN {X 0,Y 580.237,Z 574.329,A -85,B 0,C 180,E1 -1695.085,E2 -1695.085} C_VEL
LIN {X 0,Y 580.179,Z 582.821,A -85,B 0,C 180,E1 -1696.337,E2 -1696.337} C_VEL
LIN {X 0,Y 580.123,Z 588.702,A -85,B 0,C 180,E1 -1697.405,E2 -1697.405} C_VEL
LIN {X 0,Y 580.1,Z 593.511,A -85,B 0,C 180,E1 -1698.469,E2 -1698.469} C_VEL
LIN {X 0,Y 580.091,Z 598.463,A -85,B 0,C 180,E1 -1699.882,E2 -1699.882} C_VEL
LIN {X 0,Y 580.029,Z 601.153,A -85,B 0,C 180,E1 -1700.937,E2 -1700.937} C_VEL
LIN {X 0,Y 580.066,Z 603.479,A -85,B 0,C 180,E1 -1702.341,E2 -1702.341} C_VEL
LIN {X 0,Y 580.067,Z 604.438,A -85,B 0,C 180,E1 -1703.74,E2 -1703.74} C_VEL
LIN {X 0,Y 580.024,Z 604.067,A -85,B 0,C 180,E1 -1705.135,E2 -1705.135} C_VEL
LIN {X 0,Y 580.106,Z 602.365,A -85,B 0,C 180,E1 -1706.527,E2 -1706.527} C_VEL
LIN {X 0,Y 580.042,Z 599.297,A -85,B 0,C 180,E1 -1707.917,E2 -1707.917} C_VEL
LIN {X 0,Y 580.077,Z 594.788,A -85,B 0,C 180,E1 -1709.306,E2 -1709.306} C_VEL
LIN {X 0,Y 580.142,Z 590.33,A -85,B 0,C 180,E1 -1710.347,E2 -1710.347} C_VEL
LIN {X 0,Y 580.165,Z 583.928,A -85,B 0,C 180,E1 -1711.562,E2 -1711.562} C_VEL
LIN {X 0,Y 580.183,Z 576.009,A -85,B 0,C 180,E1 -1712.777,E2 -1712.777} C_VEL
LIN {X 0,Y 580.314,Z 567.745,A -85,B 0,C 180,E1 -1713.819,E2 -1713.819} C_VEL
LIN {X 0,Y 580.391,Z 557.842,A -85,B 0,C 180,E1 -1714.862,E2 -1714.862} C_VEL
LIN {X 0,Y 580.551,Z 546.821,A -85,B 0,C 180,E1 -1715.819,E2 -1715.819} C_VEL
LIN {X 0,Y 580.674,Z 535.969,A -85,B 0,C 180,E1 -1716.599,E2 -1716.599} C_VEL
LIN {X 0,Y 580.796,Z 524.77,A -85,B 0,C 180,E1 -1717.264,E2 -1717.264} C_VEL
LIN {X 0,Y 580.93,Z 511.174,A -85,B 0,C 180,E1 -1717.909,E2 -1717.909} C_VEL
LIN {X 0,Y 581.013,Z 497.115,A -85,B 0,C 180,E1 -1718.412,E2 -1718.412} C_VEL
LIN {X 0,Y 581.118,Z 483.167,A -85,B 0,C 180,E1 -1718.76,E2 -1718.76} C_VEL
LIN {X 0,Y 581.18,Z 465.651,A -85,B 0,C 180,E1 -1719.022,E2 -1719.022} C_VEL
LIN {X 0,Y 581.364,Z 347.457,A -85,B 0,C 180,E1 -1720.503,E2 -1720.503} C_VEL
LIN {X 0,Y 580.519,Z 342.708,A -85,B 0,C 180,E1 -1720.595,E2 -1720.595} C_VEL
LIN {X 0,Y 580.66,Z 323.699,A -85,B 0,C 180,E1 -1723.473,E2 -1723.473} C_VEL
LIN {X 0,Y 580.598,Z 313.228,A -85,B 0,C 180,E1 -1725.085,E2 -1725.085} C_VEL
LIN {X 0,Y 580.318,Z 311.824,A -85,B 0,C 180,E1 -1725.317,E2 -1725.317} C_VEL
LIN {X 0,Y 580.302,Z 311.826,A -85,B 0,C 180,E1 -1727.624,E2 -1727.624} C_VEL
LIN {X 0,Y 580.289,Z 311.831,A -85,B 0,C 180,E1 -1729.822,E2 -1729.822} C_VEL
LIN {X 0,Y 580.272,Z 311.831,A -85,B 0,C 180,E1 -1732.052,E2 -1732.052} C_VEL
LIN {X 0,Y 580.309,Z 311.82,A -85,B 0,C 180,E1 -1735.079,E2 -1735.079} C_VEL
LIN {X 0,Y 580.299,Z 311.823,A -85,B 0,C 180,E1 -1738.185,E2 -1738.185} C_VEL
LIN {X 0,Y 580.286,Z 311.822,A -85,B 0,C 180,E1 -1740.694,E2 -1740.694} C_VEL
LIN {X 0,Y 580.303,Z 311.824,A -85,B 0,C 180,E1 -1743.315,E2 -1743.315} C_VEL
LIN {X 0,Y 580.271,Z 311.83,A -85,B 0,C 180,E1 -1745.759,E2 -1745.759} C_VEL
LIN {X 0,Y 580.285,Z 311.823,A -85,B 0,C 180,E1 -1748.145,E2 -1748.145} C_VEL
LIN {X 0,Y 580.296,Z 311.819,A -85,B 0,C 180,E1 -1750.842,E2 -1750.842} C_VEL
LIN {X 0,Y 580.268,Z 311.83,A -85,B 0,C 180,E1 -1753.657,E2 -1753.657} C_VEL
LIN {X 0,Y 580.272,Z 311.824,A -85,B 0,C 180,E1 -1756.608,E2 -1756.608} C_VEL
LIN {X 0,Y 580.292,Z 311.827,A -85,B 0,C 180,E1 -1759.155,E2 -1759.155} C_VEL
LIN {X 0,Y 580.28,Z 311.823,A -85,B 0,C 180,E1 -1761.926,E2 -1761.926} C_VEL
LIN {X 0,Y 580.249,Z 311.826,A -85,B 0,C 180,E1 -1764.452,E2 -1764.452} C_VEL
LIN {X 0,Y 580.28,Z 311.828,A -85,B 0,C 180,E1 -1766.974,E2 -1766.974} C_VEL
LIN {X 0,Y 580.28,Z 311.827,A -85,B 0,C 180,E1 -1769.424,E2 -1769.424} C_VEL
LIN {X 0,Y 580.285,Z 311.82,A -85,B 0,C 180,E1 -1772.141,E2 -1772.141} C_VEL
LIN {X 0,Y 580.276,Z 311.83,A -85,B 0,C 180,E1 -1774.918,E2 -1774.918} C_VEL
LIN {X 0,Y 580.246,Z 311.826,A -85,B 0,C 180,E1 -1777.946,E2 -1777.946} C_VEL
LIN {X 0,Y 580.281,Z 311.83,A -85,B 0,C 180,E1 -1780.912,E2 -1780.912} C_VEL
LIN {X 0,Y 580.246,Z 311.826,A -85,B 0,C 180,E1 -1783.824,E2 -1783.824} C_VEL
LIN {X 0,Y 580.251,Z 311.833,A -85,B 0,C 180,E1 -1786.695,E2 -1786.695} C_VEL
LIN {X 0,Y 580.291,Z 311.83,A -85,B 0,C 180,E1 -1788.826,E2 -1788.826} C_VEL
LIN {X 0,Y 580.276,Z 311.823,A -85,B 0,C 180,E1 -1791.643,E2 -1791.643} C_VEL
LIN {X 0,Y 580.303,Z 311.825,A -85,B 0,C 180,E1 -1794.44,E2 -1794.44} C_VEL
LIN {X 0,Y 580.3,Z 311.821,A -85,B 0,C 180,E1 -1797.223,E2 -1797.223} C_VEL
LIN {X 0,Y 580.313,Z 311.82,A -85,B 0,C 180,E1 -1800,E2 -1800} C_VEL
LIN {X 0,Y 580.315,Z 311.822,A -85,B 0,C 180,E1 -1802.776,E2 -1802.776} C_VEL
LIN {X 0,Y 580.273,Z 311.823,A -85,B 0,C 180,E1 -1805.56,E2 -1805.56} C_VEL
LIN {X 0,Y 580.276,Z 311.832,A -85,B 0,C 180,E1 -1808.357,E2 -1808.357} C_VEL
LIN {X 0,Y 580.285,Z 311.821,A -85,B 0,C 180,E1 -1811.191,E2 -1811.191} C_VEL
LIN {X 0,Y 580.295,Z 311.826,A -85,B 0,C 180,E1 -1814.018,E2 -1814.018} C_VEL
LIN {X 0,Y 580.298,Z 311.821,A -85,B 0,C 180,E1 -1816.914,E2 -1816.914} C_VEL
LIN {X 0,Y 580.269,Z 311.828,A -85,B 0,C 180,E1 -1819.823,E2 -1819.823} C_VEL
LIN {X 0,Y 580.254,Z 311.833,A -85,B 0,C 180,E1 -1822.053,E2 -1822.053} C_VEL
LIN {X 0,Y 580.286,Z 311.821,A -85,B 0,C 180,E1 -1825.081,E2 -1825.081} C_VEL
LIN {X 0,Y 580.267,Z 311.831,A -85,B 0,C 180,E1 -1828.187,E2 -1828.187} C_VEL
LIN {X 0,Y 580.269,Z 311.824,A -85,B 0,C 180,E1 -1830.695,E2 -1830.695} C_VEL
LIN {X 0,Y 580.29,Z 311.822,A -85,B 0,C 180,E1 -1833.317,E2 -1833.317} C_VEL
LIN {X 0,Y 580.255,Z 311.834,A -85,B 0,C 180,E1 -1835.76,E2 -1835.76} C_VEL
LIN {X 0,Y 580.279,Z 311.827,A -85,B 0,C 180,E1 -1838.147,E2 -1838.147} C_VEL
LIN {X 0,Y 580.287,Z 311.82,A -85,B 0,C 180,E1 -1840.844,E2 -1840.844} C_VEL
LIN {X 0,Y 580.27,Z 311.832,A -85,B 0,C 180,E1 -1843.659,E2 -1843.659} C_VEL
LIN {X 0,Y 580.269,Z 311.824,A -85,B 0,C 180,E1 -1846.61,E2 -1846.61} C_VEL
LIN {X 0,Y 580.29,Z 311.824,A -85,B 0,C 180,E1 -1849.157,E2 -1849.157} C_VEL
LIN {X 0,Y 580.285,Z 311.826,A -85,B 0,C 180,E1 -1851.928,E2 -1851.928} C_VEL
LIN {X 0,Y 580.281,Z 311.823,A -85,B 0,C 180,E1 -1854.456,E2 -1854.456} C_VEL
LIN {X 0,Y 580.288,Z 311.825,A -85,B 0,C 180,E1 -1856.976,E2 -1856.976} C_VEL
LIN {X 0,Y 580.292,Z 311.831,A -85,B 0,C 180,E1 -1859.426,E2 -1859.426} C_VEL
LIN {X 0,Y 580.29,Z 311.822,A -85,B 0,C 180,E1 -1862.143,E2 -1862.143} C_VEL
LIN {X 0,Y 580.305,Z 311.825,A -85,B 0,C 180,E1 -1864.921,E2 -1864.921} C_VEL
LIN {X 0,Y 580.371,Z 312.027,A -85,B 0,C 180,E1 -1865.625,E2 -1865.625} C_VEL
LIN {X 0,Y 581.125,Z 316.734,A -85,B 0,C 180,E1 -1866.29,E2 -1866.29} C_VEL
LIN {X 0,Y 580.935,Z 336.517,A -85,B 0,C 180,E1 -1868.906,E2 -1868.906} C_VEL
LIN {X 0,Y 580.744,Z 359.125,A -85,B 0,C 180,E1 -1871.844,E2 -1871.844} C_VEL
LIN {X 0,Y 580.607,Z 371.577,A -85,B 0,C 180,E1 -1873.44,E2 -1873.44} C_VEL
LIN {X 0,Y 581.38,Z 377.442,A -85,B 0,C 180,E1 -1873.542,E2 -1873.542} C_VEL
LIN {X 0,Y 581.153,Z 508.664,A -85,B 0,C 180,E1 -1875.199,E2 -1875.199} C_VEL
LIN {X 0,Y 581.034,Z 523.122,A -85,B 0,C 180,E1 -1875.517,E2 -1875.517} C_VEL
LIN {X 0,Y 580.974,Z 536.209,A -85,B 0,C 180,E1 -1875.94,E2 -1875.94} C_VEL
LIN {X 0,Y 580.811,Z 549.888,A -85,B 0,C 180,E1 -1876.531,E2 -1876.531} C_VEL
LIN {X 0,Y 580.695,Z 562.69,A -85,B 0,C 180,E1 -1877.24,E2 -1877.24} C_VEL
LIN {X 0,Y 580.562,Z 574.322,A -85,B 0,C 180,E1 -1878.036,E2 -1878.036} C_VEL
LIN {X 0,Y 580.461,Z 585.969,A -85,B 0,C 180,E1 -1879.01,E2 -1879.01} C_VEL
LIN {X 0,Y 580.311,Z 596.336,A -85,B 0,C 180,E1 -1880.063,E2 -1880.063} C_VEL
LIN {X 0,Y 580.253,Z 604.914,A -85,B 0,C 180,E1 -1881.117,E2 -1881.117} C_VEL
LIN {X 0,Y 580.175,Z 613.117,A -85,B 0,C 180,E1 -1882.343,E2 -1882.343} C_VEL
LIN {X 0,Y 580.123,Z 618.992,A -85,B 0,C 180,E1 -1883.416,E2 -1883.416} C_VEL
LIN {X 0,Y 580.128,Z 623.569,A -85,B 0,C 180,E1 -1884.439,E2 -1884.439} C_VEL
LIN {X 0,Y 580.102,Z 628.443,A -85,B 0,C 180,E1 -1885.832,E2 -1885.832} C_VEL
LIN {X 0,Y 580.041,Z 631.832,A -85,B 0,C 180,E1 -1887.222,E2 -1887.222} C_VEL
LIN {X 0,Y 580.041,Z 633.832,A -85,B 0,C 180,E1 -1888.611,E2 -1888.611} C_VEL
LIN {X 0,Y 580.036,Z 634.5,A -85,B 0,C 180,E1 -1890,E2 -1890} C_VEL
LIN {X 0,Y 580.041,Z 633.833,A -85,B 0,C 180,E1 -1891.389,E2 -1891.389} C_VEL
LIN {X 0,Y 580.041,Z 631.833,A -85,B 0,C 180,E1 -1892.778,E2 -1892.778} C_VEL
LIN {X 0,Y 580.102,Z 628.444,A -85,B 0,C 180,E1 -1894.168,E2 -1894.168} C_VEL
LIN {X 0,Y 580.128,Z 623.568,A -85,B 0,C 180,E1 -1895.561,E2 -1895.561} C_VEL
LIN {X 0,Y 580.141,Z 617.053,A -85,B 0,C 180,E1 -1896.958,E2 -1896.958} C_VEL
LIN {X 0,Y 580.192,Z 609.801,A -85,B 0,C 180,E1 -1898.182,E2 -1898.182} C_VEL
LIN {X 0,Y 580.283,Z 600.825,A -85,B 0,C 180,E1 -1899.41,E2 -1899.41} C_VEL
LIN {X 0,Y 580.356,Z 591.394,A -85,B 0,C 180,E1 -1900.465,E2 -1900.465} C_VEL
LIN {X 0,Y 580.475,Z 581.323,A -85,B 0,C 180,E1 -1901.404,E2 -1901.404} C_VEL
LIN {X 0,Y 580.597,Z 569.437,A -85,B 0,C 180,E1 -1902.318,E2 -1902.318} C_VEL
LIN {X 0,Y 580.731,Z 556.653,A -85,B 0,C 180,E1 -1903.115,E2 -1903.115} C_VEL
LIN {X 0,Y 580.86,Z 544.165,A -85,B 0,C 180,E1 -1903.736,E2 -1903.736} C_VEL
LIN {X 0,Y 581.01,Z 531.19,A -85,B 0,C 180,E1 -1904.236,E2 -1904.236} C_VEL
LIN {X 0,Y 581.082,Z 517.184,A -85,B 0,C 180,E1 -1904.631,E2 -1904.631} C_VEL
LIN {X 0,Y 581.155,Z 502.632,A -85,B 0,C 180,E1 -1904.89,E2 -1904.89} C_VEL
LIN {X 0,Y 581.278,Z 375.204,A -85,B 0,C 180,E1 -1906.489,E2 -1906.489} C_VEL
LIN {X 0,Y 580.603,Z 371.489,A -85,B 0,C 180,E1 -1906.571,E2 -1906.571} C_VEL
LIN {X 0,Y 580.805,Z 350.324,A -85,B 0,C 180,E1 -1909.294,E2 -1909.294} C_VEL
LIN {X 0,Y 581.049,Z 328.038,A -85,B 0,C 180,E1 -1912.208,E2 -1912.208} C_VEL
LIN {X 0,Y 581.021,Z 315.321,A -85,B 0,C 180,E1 -1913.904,E2 -1913.904} C_VEL
LIN {X 0,Y 580.338,Z 311.825,A -85,B 0,C 180,E1 -1914.44,E2 -1914.44} C_VEL
LIN {X 0,Y 580.279,Z 311.824,A -85,B 0,C 180,E1 -1917.401,E2 -1917.401} C_VEL
LIN {X 0,Y 580.286,Z 311.823,A -85,B 0,C 180,E1 -1919.772,E2 -1919.772} C_VEL
LIN {X 0,Y 580.296,Z 311.826,A -85,B 0,C 180,E1 -1922.2,E2 -1922.2} C_VEL
LIN {X 0,Y 580.286,Z 311.828,A -85,B 0,C 180,E1 -1924.695,E2 -1924.695} C_VEL
LIN {X 0,Y 580.294,Z 311.819,A -85,B 0,C 180,E1 -1927.268,E2 -1927.268} C_VEL
LIN {X 0,Y 580.286,Z 311.829,A -85,B 0,C 180,E1 -1930.27,E2 -1930.27} C_VEL
LIN {X 0,Y 580.27,Z 311.827,A -85,B 0,C 180,E1 -1932.706,E2 -1932.706} C_VEL
LIN {X 0,Y 580.262,Z 311.825,A -85,B 0,C 180,E1 -1935.608,E2 -1935.608} C_VEL
LIN {X 0,Y 580.305,Z 311.829,A -85,B 0,C 180,E1 -1938.233,E2 -1938.233} C_VEL
LIN {X 0,Y 580.266,Z 311.825,A -85,B 0,C 180,E1 -1940.964,E2 -1940.964} C_VEL
LIN {X 0,Y 580.263,Z 311.827,A -85,B 0,C 180,E1 -1943.596,E2 -1943.596} C_VEL
LIN {X 0,Y 580.302,Z 311.828,A -85,B 0,C 180,E1 -1946.144,E2 -1946.144} C_VEL
LIN {X 0,Y 580.262,Z 311.824,A -85,B 0,C 180,E1 -1948.614,E2 -1948.614} C_VEL
LIN {X 0,Y 580.276,Z 311.821,A -85,B 0,C 180,E1 -1951.023,E2 -1951.023} C_VEL
LIN {X 0,Y 580.259,Z 311.83,A -85,B 0,C 180,E1 -1954.15,E2 -1954.15} C_VEL
LIN {X 0,Y 580.257,Z 311.827,A -85,B 0,C 180,E1 -1956.441,E2 -1956.441} C_VEL
LIN {X 0,Y 580.256,Z 311.829,A -85,B 0,C 180,E1 -1959.437,E2 -1959.437} C_VEL
LIN {X 0,Y 580.241,Z 311.835,A -85,B 0,C 180,E1 -1961.644,E2 -1961.644} C_VEL
LIN {X 0,Y 580.244,Z 311.834,A -85,B 0,C 180,E1 -1963.825,E2 -1963.825} C_VEL
LIN {X 0,Y 580.293,Z 311.825,A -85,B 0,C 180,E1 -1965.982,E2 -1965.982} C_VEL
LIN {X 0,Y 580.251,Z 311.825,A -85,B 0,C 180,E1 -1968.826,E2 -1968.826} C_VEL
LIN {X 0,Y 580.274,Z 311.831,A -85,B 0,C 180,E1 -1971.643,E2 -1971.643} C_VEL
LIN {X 0,Y 580.275,Z 311.823,A -85,B 0,C 180,E1 -1974.44,E2 -1974.44} C_VEL
LIN {X 0,Y 580.32,Z 311.824,A -85,B 0,C 180,E1 -1977.224,E2 -1977.224} C_VEL
LIN {X 0,Y 580.315,Z 311.819,A -85,B 0,C 180,E1 -1980,E2 -1980} C_VEL
LIN {X 0,Y 580.306,Z 311.82,A -85,B 0,C 180,E1 -1982.777,E2 -1982.777} C_VEL
LIN {X 0,Y 580.308,Z 311.824,A -85,B 0,C 180,E1 -1985.56,E2 -1985.56} C_VEL
LIN {X 0,Y 580.28,Z 311.822,A -85,B 0,C 180,E1 -1988.357,E2 -1988.357} C_VEL
LIN {X 0,Y 580.287,Z 311.83,A -85,B 0,C 180,E1 -1991.192,E2 -1991.192} C_VEL
LIN {X 0,Y 580.293,Z 311.821,A -85,B 0,C 180,E1 -1994.018,E2 -1994.018} C_VEL
LIN {X 0,Y 580.3,Z 311.827,A -85,B 0,C 180,E1 -1996.915,E2 -1996.915} C_VEL
LIN {X 0,Y 580.273,Z 311.823,A -85,B 0,C 180,E1 -1999.824,E2 -1999.824} C_VEL
LIN {X 0,Y 580.273,Z 311.827,A -85,B 0,C 180,E1 -2001.301,E2 -2001.301} C_VEL
LIN {X 0,Y 579.565,Z 311.914,A -85,B 0,C 180,E1 -2001.88,E2 -2001.88} C_VEL
LIN {X 0,Y 576.686,Z 312.279,A -85,B 0,C 180,E1 -2002.82,E2 -2002.82} C_VEL
LIN {X 0,Y 574.296,Z 312.571,A -85,B 0,C 180,E1 -2003.576,E2 -2003.576} C_VEL
LIN {X 0,Y 573.3,Z 312.693,A -85,B 0,C 180,E1 -2004.16,E2 -2004.16} C_VEL
LIN {X 0,Y 573.234,Z 312.702,A -85,B 0,C 180,E1 -2004.358,E2 -2004.358} C_VEL
LIN {X 0,Y 573.241,Z 312.706,A -85,B 0,C 180,E1 -2006.977,E2 -2006.977} C_VEL
LIN {X 0,Y 573.232,Z 312.701,A -85,B 0,C 180,E1 -2009.488,E2 -2009.488} C_VEL
LIN {X 0,Y 573.247,Z 312.707,A -85,B 0,C 180,E1 -2012.646,E2 -2012.646} C_VEL
LIN {X 0,Y 573.205,Z 312.706,A -85,B 0,C 180,E1 -2015.189,E2 -2015.189} C_VEL
LIN {X 0,Y 573.228,Z 312.701,A -85,B 0,C 180,E1 -2017.809,E2 -2017.809} C_VEL
LIN {X 0,Y 573.264,Z 312.705,A -85,B 0,C 180,E1 -2020.529,E2 -2020.529} C_VEL
LIN {X 0,Y 573.248,Z 312.699,A -85,B 0,C 180,E1 -2023.671,E2 -2023.671} C_VEL
LIN {X 0,Y 573.233,Z 312.707,A -85,B 0,C 180,E1 -2026.642,E2 -2026.642} C_VEL
LIN {X 0,Y 573.257,Z 312.698,A -85,B 0,C 180,E1 -2029.477,E2 -2029.477} C_VEL
LIN {X 0,Y 573.234,Z 312.709,A -85,B 0,C 180,E1 -2032.194,E2 -2032.194} C_VEL
LIN {X 0,Y 573.251,Z 312.697,A -85,B 0,C 180,E1 -2035.227,E2 -2035.227} C_VEL
LIN {X 0,Y 573.251,Z 312.703,A -85,B 0,C 180,E1 -2037.773,E2 -2037.773} C_VEL
LIN {X 0,Y 573.267,Z 312.701,A -85,B 0,C 180,E1 -2040.635,E2 -2040.635} C_VEL
LIN {X 0,Y 573.291,Z 312.798,A -85,B 0,C 180,E1 -2042.657,E2 -2042.657} C_VEL
LIN {X 0,Y 573.794,Z 317.41,A -85,B 0,C 180,E1 -2043.397,E2 -2043.397} C_VEL
LIN {X 0,Y 573.594,Z 335.264,A -85,B 0,C 180,E1 -2046.151,E2 -2046.151} C_VEL
LIN {X 0,Y 573.504,Z 342.753,A -85,B 0,C 180,E1 -2047.294,E2 -2047.294} C_VEL
LIN {X 0,Y 574.6,Z 349.299,A -85,B 0,C 180,E1 -2047.411,E2 -2047.411} C_VEL
LIN {X 0,Y 574.271,Z 479.303,A -85,B 0,C 180,E1 -2049.074,E2 -2049.074} C_VEL
LIN {X 0,Y 574.181,Z 493.519,A -85,B 0,C 180,E1 -2049.397,E2 -2049.397} C_VEL
LIN {X 0,Y 574.036,Z 507.401,A -85,B 0,C 180,E1 -2049.859,E2 -2049.859} C_VEL
LIN {X 0,Y 573.887,Z 520.537,A -85,B 0,C 180,E1 -2050.443,E2 -2050.443} C_VEL
LIN {X 0,Y 573.736,Z 533.063,A -85,B 0,C 180,E1 -2051.151,E2 -2051.151} C_VEL
LIN {X 0,Y 573.563,Z 544.908,A -85,B 0,C 180,E1 -2051.978,E2 -2051.978} C_VEL
LIN {X 0,Y 573.395,Z 556.302,A -85,B 0,C 180,E1 -2052.948,E2 -2052.948} C_VEL
LIN {X 0,Y 573.274,Z 566.375,A -85,B 0,C 180,E1 -2053.989,E2 -2053.989} C_VEL
LIN {X 0,Y 573.175,Z 575.123,A -85,B 0,C 180,E1 -2055.079,E2 -2055.079} C_VEL
LIN {X 0,Y 573.116,Z 583.422,A -85,B 0,C 180,E1 -2056.346,E2 -2056.346} C_VEL
LIN {X 0,Y 573.037,Z 590.065,A -85,B 0,C 180,E1 -2057.607,E2 -2057.607} C_VEL
LIN {X 0,Y 573.046,Z 595.28,A -85,B 0,C 180,E1 -2058.858,E2 -2058.858} C_VEL
LIN {X 0,Y 573,Z 599.266,A -85,B 0,C 180,E1 -2060.113,E2 -2060.113} C_VEL
LIN {X 0,Y 572.951,Z 602.371,A -85,B 0,C 180,E1 -2061.536,E2 -2061.536} C_VEL
LIN {X 0,Y 572.971,Z 604.076,A -85,B 0,C 180,E1 -2062.955,E2 -2062.955} C_VEL
LIN {X 0,Y 572.991,Z 604.435,A -85,B 0,C 180,E1 -2064.369,E2 -2064.369} C_VEL
LIN {X 0,Y 573.005,Z 603.466,A -85,B 0,C 180,E1 -2065.78,E2 -2065.78} C_VEL
LIN {X 0,Y 572.953,Z 601.157,A -85,B 0,C 180,E1 -2067.188,E2 -2067.188} C_VEL
LIN {X 0,Y 572.965,Z 597.453,A -85,B 0,C 180,E1 -2068.594,E2 -2068.594} C_VEL
LIN {X 0,Y 573.007,Z 592.26,A -85,B 0,C 180,E1 -2070,E2 -2070} C_VEL
LIN {X 0,Y 573.086,Z 587.233,A -85,B 0,C 180,E1 -2071.054,E2 -2071.054} C_VEL
LIN {X 0,Y 573.117,Z 580.087,A -85,B 0,C 180,E1 -2072.284,E2 -2072.284} C_VEL
LIN {X 0,Y 573.236,Z 572.626,A -85,B 0,C 180,E1 -2073.338,E2 -2073.338} C_VEL
LIN {X 0,Y 573.341,Z 563.699,A -85,B 0,C 180,E1 -2074.394,E2 -2074.394} C_VEL
LIN {X 0,Y 573.47,Z 552.935,A -85,B 0,C 180,E1 -2075.45,E2 -2075.45} C_VEL
LIN {X 0,Y 573.615,Z 542.04,A -85,B 0,C 180,E1 -2076.331,E2 -2076.331} C_VEL
LIN {X 0,Y 573.763,Z 529.263,A -85,B 0,C 180,E1 -2077.172,E2 -2077.172} C_VEL
LIN {X 0,Y 573.943,Z 516.796,A -85,B 0,C 180,E1 -2077.829,E2 -2077.829} C_VEL
LIN {X 0,Y 574.121,Z 502.712,A -85,B 0,C 180,E1 -2078.403,E2 -2078.403} C_VEL
LIN {X 0,Y 574.25,Z 489.376,A -85,B 0,C 180,E1 -2078.8,E2 -2078.8} C_VEL
LIN {X 0,Y 574.319,Z 474.642,A -85,B 0,C 180,E1 -2079.087,E2 -2079.087} C_VEL
LIN {X 0,Y 574.479,Z 347.892,A -85,B 0,C 180,E1 -2080.701,E2 -2080.701} C_VEL
LIN {X 0,Y 573.557,Z 342.696,A -85,B 0,C 180,E1 -2080.803,E2 -2080.803} C_VEL
LIN {X 0,Y 573.718,Z 324.206,A -85,B 0,C 180,E1 -2083.639,E2 -2083.639} C_VEL
LIN {X 0,Y 573.686,Z 314.898,A -85,B 0,C 180,E1 -2085.089,E2 -2085.089} C_VEL
LIN {X 0,Y 573.277,Z 312.702,A -85,B 0,C 180,E1 -2085.464,E2 -2085.464} C_VEL
LIN {X 0,Y 573.254,Z 312.707,A -85,B 0,C 180,E1 -2087.848,E2 -2087.848} C_VEL
LIN {X 0,Y 573.244,Z 312.707,A -85,B 0,C 180,E1 -2090.076,E2 -2090.076} C_VEL
LIN {X 0,Y 573.236,Z 312.703,A -85,B 0,C 180,E1 -2092.337,E2 -2092.337} C_VEL
LIN {X 0,Y 573.257,Z 312.701,A -85,B 0,C 180,E1 -2095.409,E2 -2095.409} C_VEL
LIN {X 0,Y 573.252,Z 312.703,A -85,B 0,C 180,E1 -2098.028,E2 -2098.028} C_VEL
LIN {X 0,Y 573.232,Z 312.701,A -85,B 0,C 180,E1 -2100.882,E2 -2100.882} C_VEL
LIN {X 0,Y 573.262,Z 312.704,A -85,B 0,C 180,E1 -2103.523,E2 -2103.523} C_VEL
LIN {X 0,Y 573.241,Z 312.702,A -85,B 0,C 180,E1 -2106.048,E2 -2106.048} C_VEL
LIN {X 0,Y 573.245,Z 312.699,A -85,B 0,C 180,E1 -2108.7,E2 -2108.7} C_VEL
LIN {X 0,Y 573.227,Z 312.709,A -85,B 0,C 180,E1 -2111.592,E2 -2111.592} C_VEL
LIN {X 0,Y 573.224,Z 312.701,A -85,B 0,C 180,E1 -2114.333,E2 -2114.333} C_VEL
LIN {X 0,Y 573.236,Z 312.71,A -85,B 0,C 180,E1 -2117.357,E2 -2117.357} C_VEL
LIN {X 0,Y 573.233,Z 312.7,A -85,B 0,C 180,E1 -2120.391,E2 -2120.391} C_VEL
LIN {X 0,Y 573.245,Z 312.704,A -85,B 0,C 180,E1 -2123.076,E2 -2123.076} C_VEL
LIN {X 0,Y 573.257,Z 312.699,A -85,B 0,C 180,E1 -2125.67,E2 -2125.67} C_VEL
LIN {X 0,Y 573.236,Z 312.699,A -85,B 0,C 180,E1 -2128.184,E2 -2128.184} C_VEL
LIN {X 0,Y 573.248,Z 312.701,A -85,B 0,C 180,E1 -2130.633,E2 -2130.633} C_VEL
LIN {X 0,Y 573.239,Z 312.706,A -85,B 0,C 180,E1 -2133.023,E2 -2133.023} C_VEL
LIN {X 0,Y 573.223,Z 312.706,A -85,B 0,C 180,E1 -2135.363,E2 -2135.363} C_VEL
LIN {X 0,Y 573.214,Z 312.703,A -85,B 0,C 180,E1 -2137.661,E2 -2137.661} C_VEL
LIN {X 0,Y 573.253,Z 312.701,A -85,B 0,C 180,E1 -2140.669,E2 -2140.669} C_VEL
LIN {X 0,Y 573.223,Z 312.702,A -85,B 0,C 180,E1 -2143.621,E2 -2143.621} C_VEL
LIN {X 0,Y 573.208,Z 312.707,A -85,B 0,C 180,E1 -2146.529,E2 -2146.529} C_VEL
LIN {X 0,Y 573.248,Z 312.705,A -85,B 0,C 180,E1 -2148.745,E2 -2148.745} C_VEL
LIN {X 0,Y 573.223,Z 312.702,A -85,B 0,C 180,E1 -2151.539,E2 -2151.539} C_VEL
LIN {X 0,Y 573.195,Z 312.704,A -85,B 0,C 180,E1 -2153.664,E2 -2153.664} C_VEL
LIN {X 0,Y 573.18,Z 312.704,A -85,B 0,C 180,E1 -2155.781,E2 -2155.781} C_VEL
LIN {X 0,Y 573.271,Z 312.695,A -85,B 0,C 180,E1 -2157.892,E2 -2157.892} C_VEL
LIN {X 0,Y 573.316,Z 312.697,A -85,B 0,C 180,E1 -2160.702,E2 -2160.702} C_VEL
LIN {X 0,Y 573.278,Z 312.698,A -85,B 0,C 180,E1 -2162.811,E2 -2162.811} C_VEL
LIN {X 0,Y 573.243,Z 312.699,A -85,B 0,C 180,E1 -2165.628,E2 -2165.628} C_VEL
LIN {X 0,Y 573.222,Z 312.709,A -85,B 0,C 180,E1 -2168.46,E2 -2168.46} C_VEL
LIN {X 0,Y 573.257,Z 312.697,A -85,B 0,C 180,E1 -2171.312,E2 -2171.312} C_VEL
LIN {X 0,Y 573.259,Z 312.703,A -85,B 0,C 180,E1 -2174.421,E2 -2174.421} C_VEL
LIN {X 0,Y 573.24,Z 312.699,A -85,B 0,C 180,E1 -2177.112,E2 -2177.112} C_VEL
LIN {X 0,Y 573.225,Z 312.709,A -85,B 0,C 180,E1 -2180.077,E2 -2180.077} C_VEL
LIN {X 0,Y 573.217,Z 312.708,A -85,B 0,C 180,E1 -2182.338,E2 -2182.338} C_VEL
LIN {X 0,Y 573.231,Z 312.701,A -85,B 0,C 180,E1 -2185.411,E2 -2185.411} C_VEL
LIN {X 0,Y 573.213,Z 312.704,A -85,B 0,C 180,E1 -2188.566,E2 -2188.566} C_VEL
LIN {X 0,Y 573.212,Z 312.702,A -85,B 0,C 180,E1 -2190.994,E2 -2190.994} C_VEL
LIN {X 0,Y 573.252,Z 312.702,A -85,B 0,C 180,E1 -2193.525,E2 -2193.525} C_VEL
LIN {X 0,Y 573.23,Z 312.707,A -85,B 0,C 180,E1 -2196.05,E2 -2196.05} C_VEL
LIN {X 0,Y 573.232,Z 312.7,A -85,B 0,C 180,E1 -2198.702,E2 -2198.702} C_VEL
LIN {X 0,Y 573.243,Z 312.705,A -85,B 0,C 180,E1 -2201.596,E2 -2201.596} C_VEL
LIN {X 0,Y 573.227,Z 312.702,A -85,B 0,C 180,E1 -2204.334,E2 -2204.334} C_VEL
LIN {X 0,Y 573.233,Z 312.705,A -85,B 0,C 180,E1 -2207.359,E2 -2207.359} C_VEL
LIN {X 0,Y 573.235,Z 312.701,A -85,B 0,C 180,E1 -2210.393,E2 -2210.393} C_VEL
LIN {X 0,Y 573.25,Z 312.702,A -85,B 0,C 180,E1 -2213.079,E2 -2213.079} C_VEL
LIN {X 0,Y 573.264,Z 312.704,A -85,B 0,C 180,E1 -2215.672,E2 -2215.672} C_VEL
LIN {X 0,Y 573.238,Z 312.701,A -85,B 0,C 180,E1 -2218.185,E2 -2218.185} C_VEL
LIN {X 0,Y 573.263,Z 312.698,A -85,B 0,C 180,E1 -2220.635,E2 -2220.635} C_VEL
LIN {X 0,Y 573.235,Z 312.709,A -85,B 0,C 180,E1 -2223.508,E2 -2223.508} C_VEL
LIN {X 0,Y 573.297,Z 312.727,A -85,B 0,C 180,E1 -2225.416,E2 -2225.416} C_VEL
LIN {X 0,Y 574.25,Z 318.109,A -85,B 0,C 180,E1 -2226.18,E2 -2226.18} C_VEL
LIN {X 0,Y 574.018,Z 338.181,A -85,B 0,C 180,E1 -2228.861,E2 -2228.861} C_VEL
LIN {X 0,Y 573.786,Z 360.538,A -85,B 0,C 180,E1 -2231.8,E2 -2231.8} C_VEL
LIN {X 0,Y 573.638,Z 371.699,A -85,B 0,C 180,E1 -2233.24,E2 -2233.24} C_VEL
LIN {X 0,Y 574.573,Z 377.498,A -85,B 0,C 180,E1 -2233.342,E2 -2233.342} C_VEL
LIN {X 0,Y 574.304,Z 508.663,A -85,B 0,C 180,E1 -2235.018,E2 -2235.018} C_VEL
LIN {X 0,Y 574.152,Z 523.411,A -85,B 0,C 180,E1 -2235.348,E2 -2235.348} C_VEL
LIN {X 0,Y 574.023,Z 537.72,A -85,B 0,C 180,E1 -2235.826,E2 -2235.826} C_VEL
LIN {X 0,Y 573.869,Z 551.651,A -85,B 0,C 180,E1 -2236.455,E2 -2236.455} C_VEL
LIN {X 0,Y 573.718,Z 564.107,A -85,B 0,C 180,E1 -2237.172,E2 -2237.172} C_VEL
LIN {X 0,Y 573.532,Z 576.647,A -85,B 0,C 180,E1 -2238.066,E2 -2238.066} C_VEL
LIN {X 0,Y 573.436,Z 588.18,A -85,B 0,C 180,E1 -2239.084,E2 -2239.084} C_VEL
LIN {X 0,Y 573.239,Z 597.854,A -85,B 0,C 180,E1 -2240.117,E2 -2240.117} C_VEL
LIN {X 0,Y 573.202,Z 606.174,A -85,B 0,C 180,E1 -2241.184,E2 -2241.184} C_VEL
LIN {X 0,Y 573.11,Z 614.128,A -85,B 0,C 180,E1 -2242.425,E2 -2242.425} C_VEL
LIN {X 0,Y 573.02,Z 620.528,A -85,B 0,C 180,E1 -2243.663,E2 -2243.663} C_VEL
LIN {X 0,Y 573.001,Z 624.962,A -85,B 0,C 180,E1 -2244.722,E2 -2244.722} C_VEL
LIN {X 0,Y 573.028,Z 628.443,A -85,B 0,C 180,E1 -2245.78,E2 -2245.78} C_VEL
LIN {X 0,Y 572.956,Z 631.832,A -85,B 0,C 180,E1 -2247.188,E2 -2247.188} C_VEL
LIN {X 0,Y 572.941,Z 633.833,A -85,B 0,C 180,E1 -2248.594,E2 -2248.594} C_VEL
LIN {X 0,Y 572.937,Z 634.5,A -85,B 0,C 180,E1 -2250,E2 -2250} C_VEL
LIN {X 0,Y 572.941,Z 633.833,A -85,B 0,C 180,E1 -2251.406,E2 -2251.406} C_VEL
LIN {X 0,Y 572.956,Z 631.834,A -85,B 0,C 180,E1 -2252.812,E2 -2252.812} C_VEL
LIN {X 0,Y 573.028,Z 628.445,A -85,B 0,C 180,E1 -2254.22,E2 -2254.22} C_VEL
LIN {X 0,Y 573.059,Z 623.569,A -85,B 0,C 180,E1 -2255.63,E2 -2255.63} C_VEL
LIN {X 0,Y 573.058,Z 618.852,A -85,B 0,C 180,E1 -2256.693,E2 -2256.693} C_VEL
LIN {X 0,Y 573.125,Z 612.038,A -85,B 0,C 180,E1 -2257.929,E2 -2257.929} C_VEL
LIN {X 0,Y 573.225,Z 603.56,A -85,B 0,C 180,E1 -2259.171,E2 -2259.171} C_VEL
LIN {X 0,Y 573.304,Z 594.71,A -85,B 0,C 180,E1 -2260.239,E2 -2260.239} C_VEL
LIN {X 0,Y 573.461,Z 583.994,A -85,B 0,C 180,E1 -2261.308,E2 -2261.308} C_VEL
LIN {X 0,Y 573.616,Z 573.146,A -85,B 0,C 180,E1 -2262.201,E2 -2262.201} C_VEL
LIN {X 0,Y 573.74,Z 561.263,A -85,B 0,C 180,E1 -2263.007,E2 -2263.007} C_VEL
LIN {X 0,Y 573.945,Z 548.103,A -85,B 0,C 180,E1 -2263.724,E2 -2263.724} C_VEL
LIN {X 0,Y 574.085,Z 534.827,A -85,B 0,C 180,E1 -2264.284,E2 -2264.284} C_VEL
LIN {X 0,Y 574.204,Z 520.758,A -85,B 0,C 180,E1 -2264.721,E2 -2264.721} C_VEL
LIN {X 0,Y 574.302,Z 507.158,A -85,B 0,C 180,E1 -2265.004,E2 -2265.004} C_VEL
LIN {X 0,Y 574.532,Z 376.416,A -85,B 0,C 180,E1 -2266.673,E2 -2266.673} C_VEL
